# B&R Automation Studio project LABA4FINAL
Automation Studio 

## Configuration Real

### Task classes (Cpu.sw)
```
Cyclic#1:
  ncsdcctrl <- ncsdcctrl.prg
  SDCAxisCtr <- SDCAxisCtr.prg
  SDCAxisCt1 <- SDCAxisCtr1.prg
  SDCAxisCt2 <- SDCAxisCtr2.prg
DataObjects: Arnc0sys
NcDataObjects: AxisInit <- AxisInit.dob, gAxis03a <- gAxis03obj.gAxis03a.dob, gAxis03i <- gAxis03obj.gAxis03i.dob, AxisApt <- AxisApt.dob, gmcipvar <- GmcIpUserConfig.gmcipvar.dob, gmcipfun <- GmcIpUserConfig.gmcipfun.dob, gmcipfub <- GmcIpUserConfig.gmcipfub.dob, gmcipubr <- GmcIpUserConfig.gmcipubr.dob, gmcipusm <- GmcIpUserConfig.gmcipusm.dob, gmcipui <- GmcIpUserConfig.gmcipui.dob, gmcipus <- GmcIpUserConfig.gmcipus.dob, gmcipuc <- GmcIpUserConfig.gmcipuc.dob, gmcipsys <- GmcIpConfig.gmcipsys.dob, gmciplbr <- GmcIpConfig.gmciplbr.dob, gmcipcbr <- GmcIpConfig.gmcipcbr.dob, gmciplsm <- GmcIpConfig.gmciplsm.dob, gmcipcsm <- GmcIpConfig.gmcipcsm.dob, gmcipcfg <- GmcIpConfig.gmcipcfg.dob, gmcipiec <- GmcIpConfig.gmcipiec.dob, gmciplog <- GmcIpConfig.gmciplog.dob, gmcipesm <- GmcIpConfig.gmcipesm.dob, gmcipmxd <- GmcIpConfig.gmcipmxd.dob, gmcipmx <- GmcIpConfig.gmcipmx.dob, CncInit <- CncInit.dob, CncProg <- CncProg.dob, CncProg1 <- CncProg1.dob
Binaries: TCData, Acp10map1, acp10cfg, Acp10map, arconfig, User, Role, sysconf, iomap, asfw, ashwd, arnc0cfg, Arnc0map
Libraries: Acp10sdc, Library, Acp10man, Acp10_MC, sys_lib, brsystem, asstring, powerlnk, asieccon, AsMath, Arnc0man, DataObj, AsArLog, FileIO, AsArProf, AsMem, Runtime, astime, Acp10par, NcGlobal, asiotime
```

### IoMap.iom - 4PP065_0571_P74/IoMap.iom
```iecst
VAR_CONFIG
	Cyclic#1.gAxis03_DrvIf.iLifeCnt AT %IB."8I64xxxxxxx.00x-1".SDC_LifeCnt;
	Cyclic#1.gAxis03_DrvIf.iDrvOK AT %IX."8I64xxxxxxx.00x-1".ETAD_Input_Bool_02;
	Cyclic#1.gAxis03_DrvIf.oSetTime AT %QW."8I64xxxxxxx.00x-1".SDC_SetTime;
	Cyclic#1.gAxis03_DrvIf.oSetPos AT %QW."8I64xxxxxxx.00x-1".LFRD_Output;
	Cyclic#1.gAxis03_DiDoIf.iLifeCntDriveReady AT %IB."8I64xxxxxxx.00x-1".SDC_LifeCnt;
	Cyclic#1.gAxis03_DiDoIf.iLifeCntDriveEnable AT %IB."8I64xxxxxxx.00x-1".SDC_LifeCnt;
	Cyclic#1.gAxis03_DiDoIf.oDriveEnable AT %QX."8I64xxxxxxx.00x-1".CMDD_Output_Bool_00;
	Cyclic#1.gAxis03_ModuleOk AT %QX."8I64xxxxxxx.00x-1".CMDD_Output_Bool_01;
	Cyclic#1.gAxis03_ModuleOk AT %QX."8I64xxxxxxx.00x-1".CMDD_Output_Bool_02;
	Cyclic#1.gAxis03_ModuleOk AT %IX."8I64xxxxxxx.00x-1".ModuleOk;
	Cyclic#1.gAxis03_DiDoIf.oDriveEnable AT %QX."8I64xxxxxxx.00x-1".CMDD_Output_Bool_03;
	Cyclic#1.gAxis03_DiDoIf.iDriveReady AT %IX."8I64xxxxxxx.00x-1".ETAD_Input_Bool_02;
	::SDCAxisCtr:pwm_period AT %QW."X20MM4456".PeriodDurationPWM;
	::SDCAxisCtr:coil_pwm_value AT %QW."X20MM4456".PulseWidthCurrentPWM04;
	::SDCAxisCtr:axis_X.pwm_value AT %QW."X20MM4456".PulseWidthCurrentPWM01;
	::SDCAxisCtr:axis_X.reset_error AT %QX."X20MM4456".ClearError01;
	::SDCAxisCtr:axis_X.reset_counter AT %QX."X20MM4456".ResetCounter01;
	::SDCAxisCtr:axis_X.counter AT %IW."X20MM4456".Counter01;
	::SDCAxisCtr:axis_X.endswitch_a_reached AT %IX."X20MM4456".StatusInput03; (*Logical condition input 01=Motor 01:A*)
	::SDCAxisCtr:axis_X.endswitch_b_reached AT %IX."X20MM4456".StatusInput04; (*Logical condition input 02=Motor 01:B*)
	::SDCAxisCtr:coil_powered AT %IX."X20DI9371".DigitalInput01;
	::SDCAxisCt1:axis_Y.pwm_value AT %QW."X20MM4456".PulseWidthCurrentPWM02;
	::SDCAxisCt1:axis_Y.reset_error AT %QX."X20MM4456".ClearError02;
	::SDCAxisCt1:axis_Y.reset_counter AT %QX."X20MM4456".ResetCounter02;
	::SDCAxisCt1:axis_Y.counter AT %IW."X20MM4456".Counter02;
	::SDCAxisCt1:axis_Y.endswitch_a_reached AT %IX."X20MM4456".StatusInput07;
	::SDCAxisCt1:axis_Y.endswitch_b_reached AT %IX."X20MM4456".StatusInput08;
	::SDCAxisCt2:axis_Z.pwm_value AT %QW."X20MM4456".PulseWidthCurrentPWM03;
	::SDCAxisCt2:axis_Z.reset_error AT %QX."X20MM4456".ClearError03;
	::SDCAxisCt2:axis_Z.reset_counter AT %QX."X20MM4456".ResetCounter03;
	::SDCAxisCt2:axis_Z.counter AT %IW."X20MM4456".Counter03;
	::SDCAxisCt2:axis_Z.endswitch_a_reached AT %IX."X20MM4456".StatusInput11;
	::SDCAxisCt2:axis_Z.endswitch_b_reached AT %IX."X20MM4456".StatusInput12;
	::SDCAxisCt1:coil_powered AT %IX."X20DI9371".DigitalInput02;
	::SDCAxisCt2:coil_powered AT %IX."X20DI9371".DigitalInput03;
END_VAR
```

### Acp10map.ncm - 4PP065_0571_P74/Motion/Acp10map.ncm
```
NcMapping (NcSwId=Acp10, DisabledNodesAreHidden=False)
  NcObject gAxis03 (ModuleId=8I64xxxxxxx.00x-1, ModuleAddress=SDC_IF1.ST1, Type=ncAXIS, Channel=1, AcoposSimulation=Off, InitParameter=gAxis03i, AcoposParameter=gAxis03a, AdditionalData=CNC_Enabled="1" , Disabled=FALSE, ModuleDisabled=FALSE)
```

### Arnc0map.ncm - 4PP065_0571_P74/Motion/Arnc0map.ncm
```
NcMapping (NcSwId=Arnc0, DisabledNodesAreHidden=False)
  NcObject CNCsys (Type=ncCNCSYS, Channel=1, AcoposSimulation=Off, InitParameter=CncInit, Disabled=FALSE, ModuleDisabled=FALSE)
  NcObject CNC2 (Type=ncCNCSYS, Channel=2, AcoposSimulation=Off, Disabled=TRUE, ModuleDisabled=FALSE)
  NcObject CNC3 (Type=ncCNCSYS, Channel=3, AcoposSimulation=Off, Disabled=TRUE, ModuleDisabled=FALSE)
  NcObject CNC4 (Type=ncCNCSYS, Channel=4, AcoposSimulation=Off, Disabled=TRUE, ModuleDisabled=FALSE)
  NcObject CNC5 (Type=ncCNCSYS, Channel=5, AcoposSimulation=Off, Disabled=TRUE, ModuleDisabled=FALSE)
  NcObject CNC6 (Type=ncCNCSYS, Channel=6, AcoposSimulation=Off, Disabled=TRUE, ModuleDisabled=FALSE)
  NcObject CNC7 (Type=ncCNCSYS, Channel=7, AcoposSimulation=Off, Disabled=TRUE, ModuleDisabled=FALSE)
  NcObject CNC8 (Type=ncCNCSYS, Channel=8, AcoposSimulation=Off, Disabled=TRUE, ModuleDisabled=FALSE)
  NcObject CNC9 (Type=ncCNCSYS, Channel=9, AcoposSimulation=Off, Disabled=TRUE, ModuleDisabled=FALSE)
  NcObject CNC10 (Type=ncCNCSYS, Channel=10, AcoposSimulation=Off, Disabled=TRUE, ModuleDisabled=FALSE)
  NcObject CNC11 (Type=ncCNCSYS, Channel=11, AcoposSimulation=Off, Disabled=TRUE, ModuleDisabled=FALSE)
  NcObject CNC12 (Type=ncCNCSYS, Channel=12, AcoposSimulation=Off, Disabled=TRUE, ModuleDisabled=FALSE)
  NcObject CNC13 (Type=ncCNCSYS, Channel=13, AcoposSimulation=Off, Disabled=TRUE, ModuleDisabled=FALSE)
  NcObject CNC14 (Type=ncCNCSYS, Channel=14, AcoposSimulation=Off, Disabled=TRUE, ModuleDisabled=FALSE)
  NcObject CNC15 (Type=ncCNCSYS, Channel=15, AcoposSimulation=Off, Disabled=TRUE, ModuleDisabled=FALSE)
  NcObject CNC16 (Type=ncCNCSYS, Channel=16, AcoposSimulation=Off, Disabled=TRUE, ModuleDisabled=FALSE)
  NcObject CNC17 (Type=ncCNCSYS, Channel=17, AcoposSimulation=Off, Disabled=TRUE, ModuleDisabled=FALSE)
  NcObject CNC18 (Type=ncCNCSYS, Channel=18, AcoposSimulation=Off, Disabled=TRUE, ModuleDisabled=FALSE)
  NcObject CNC19 (Type=ncCNCSYS, Channel=19, AcoposSimulation=Off, Disabled=TRUE, ModuleDisabled=FALSE)
  NcObject CNC20 (Type=ncCNCSYS, Channel=20, AcoposSimulation=Off, Disabled=TRUE, ModuleDisabled=FALSE)
  NcObject CNC21 (Type=ncCNCSYS, Channel=21, AcoposSimulation=Off, Disabled=TRUE, ModuleDisabled=FALSE)
  NcObject CNC22 (Type=ncCNCSYS, Channel=22, AcoposSimulation=Off, Disabled=TRUE, ModuleDisabled=FALSE)
  NcObject CNC23 (Type=ncCNCSYS, Channel=23, AcoposSimulation=Off, Disabled=TRUE, ModuleDisabled=FALSE)
  NcObject CNC24 (Type=ncCNCSYS, Channel=24, AcoposSimulation=Off, Disabled=TRUE, ModuleDisabled=FALSE)
```

## Configuration Simulation

CPU , AutomationRuntime J4.25

### Task classes (Cpu.sw)
```
Cyclic#1 (cycle 100000 us, tolerance 0 us):
  SDCAxisCtr <- SDCAxisCtr.prg
DataObjects: Acp10sys
NcDataObjects: AxisApt <- AxisApt.dob, AxisInit <- AxisInit.dob, acp10etxen <- acp10etxen.dob
Binaries: TCData, ashwd, sysconf, asfw, arconfig, iomap, Acp10map, Acp10map1, arnc0cfg, acp10cfg
Libraries: AsIecCon, astime, Acp10sdc, Acp10man, Acp10par, NcGlobal, asstring, AsIOTime, Acp10_MC, brsystem, sys_lib, Runtime, Acp10sim, fileio, powerlnk, Library
```

### Hardware
```
PC_any : PC_any v1.1.0.0 (OrderNumber=PC)
  ConfigurationID = SDCAxis_Simulation
  Cyclic1Duration = 100000
  Cyclic1Tolerance = 0
  Cyclic2Duration = 200000
  Cyclic2Tolerance = 10000000
  Cyclic3Duration = 500000
  Cyclic3Tolerance = 10000000
  Cyclic4Duration = 1000000
  Cyclic4Tolerance = 10000000
  Cyclic5Duration = 2000000
  Cyclic5Tolerance = 10000000
  Cyclic6Duration = 3000000
  Cyclic6Tolerance = 12000000
  Cyclic7Duration = 4000000
  Cyclic7Tolerance = 12000000
  Cyclic8Duration = 5000000
  Cyclic8Tolerance = 30000000
```

## Logical view

### Global.var - Global variables
```iecst
VAR
	AxisX : ACP10AXIS_typ := (0);
	AxisX_EncIf : SdcEncIf16_typ := (0);
	AxisX_DrvIf : SdcDrvIf16_typ := (0);
	AxisX_DiDoIf : SdcDiDoIf_typ := (0);
	AxisX_HW : SdcHwCfg_typ := (0);
	AxisY : ACP10AXIS_typ := (0);
	AxisY_EncIf : SdcEncIf16_typ := (0);
	AxisY_DrvIf : SdcDrvIf16_typ := (0);
	AxisY_DiDoIf : SdcDiDoIf_typ := (0);
	AxisY_HW : SdcHwCfg_typ := (0);
	AxisZ : ACP10AXIS_typ := (0);
	AxisZ_EncIf : SdcEncIf16_typ := (0);
	AxisZ_DrvIf : SdcDrvIf16_typ := (0);
	AxisZ_DiDoIf : SdcDiDoIf_typ := (0);
	AxisZ_HW : SdcHwCfg_typ := (0);
	gAxis01 : ACP10AXIS_typ := (0);
	gAxis02 : ACP10AXIS_typ := (0);
	gAxisTest : ACP10AXIS_typ := (0);
	gAxisTest_HW : SdcHwCfg_typ := (0);
	gAxisTest_DrvIf : SdcDrvIf16_typ := (0);
	gAxisTest_DiDoIf : SdcDiDoIf_typ := (0);
	gAxisTest_ModuleOk : BOOL := 0;
	gAxis03 : ACP10AXIS_typ := (0);
	gAxis03_HW : SdcHwCfg_typ := (0);
	gAxis03_DrvIf : SdcDrvIf16_typ := (0);
	gAxis03_DiDoIf : SdcDiDoIf_typ := (0);
	gAxis03_ModuleOk : BOOL := 0;
	CNCsys : ARNC0CNC_typ;
END_VAR
```

### Package Logical/Libraries - Global libraries

### Library Logical/Libraries/Library (ANSIC)

#### Library.fun
```iecst
FUNCTION_BLOCK FB_Motor (*TODO: Add your comment here*) (*$GROUP=User,$CAT=User,$GROUPICON=User.png,$CATICON=User.png*)
	VAR_INPUT
		in : REAL;
	END_VAR
	VAR_OUTPUT
		out_w : REAL;
		out_phi : REAL;
	END_VAR
	VAR
		k_e : REAL;
		T_m : REAL;
		dt : REAL;
		integrator : FB_Integrator;
		integrator_phi : FB_Integrator;
	END_VAR
END_FUNCTION_BLOCK

FUNCTION_BLOCK FB_Integrator (*TODO: Add your comment here*) (*$GROUP=User,$CAT=User,$GROUPICON=User.png,$CATICON=User.png*)
	VAR_INPUT
		in : REAL;
		dt : REAL;
	END_VAR
	VAR_OUTPUT
		out : REAL;
	END_VAR
	VAR
		state : REAL := 0.0;
	END_VAR
END_FUNCTION_BLOCK

FUNCTION_BLOCK FB_Controller (* *) (*$GROUP=User,$CAT=User,$GROUPICON=User.png,$CATICON=User.png*)
	VAR_INPUT
		in : REAL;
	END_VAR
	VAR_OUTPUT
		out : REAL;
	END_VAR
	VAR
		k_i : REAL;
		sum : REAL;
		k_p : REAL;
		dt : REAL;
		max_abs_value : REAL;
		integrator : FB_Integrator;
		last_sum : REAL;
	END_VAR
END_FUNCTION_BLOCK

FUNCTION_BLOCK FB_Endswitch (*TODO: Add your comment here*) (*$GROUP=User,$CAT=User,$GROUPICON=User.png,$CATICON=User.png*)
	VAR_INPUT
		in : REAL;
		neg_value : REAL;
		pos_value : REAL;
	END_VAR
	VAR_OUTPUT
		neg_reached : BOOL;
		pos_reached : BOOL;
	END_VAR
END_FUNCTION_BLOCK

FUNCTION_BLOCK FB_Axis (*TODO: Add your comment here*) (*$GROUP=User,$CAT=User,$GROUPICON=User.png,$CATICON=User.png*)
	VAR_INPUT
		reset_error : BOOL;
		endswitch_a_reached : BOOL;
		endswitch_b_reached : BOOL;
		pwm_percentage : SINT;
	END_VAR
	VAR_OUTPUT
		reset_counter : BOOL;
		pwm_value : INT;
	END_VAR
	VAR_OUTPUT RETAIN
		counter : INT;
	END_VAR
	VAR_OUTPUT
		speed : REAL;
	END_VAR
	VAR
		last_counter : INT;
	END_VAR
END_FUNCTION_BLOCK
```

#### FB_Controller.c
```c
#include <bur/plctypes.h>
#ifdef __cplusplus
	extern "C"
	{
#endif
	#include "Library.h"
#ifdef __cplusplus
	};
#endif

void FB_Controller(struct FB_Controller* inst)
{
	REAL a = inst->in * inst->k_p;
	REAL b = inst->in * inst->k_i;
	inst->integrator.dt = inst->dt;
	inst->integrator.in = b;
	FB_Integrator(&inst->integrator);
	a = a > inst->max_abs_value ? inst->max_abs_value : a;
	a = a < -inst->max_abs_value ? -inst->max_abs_value : a;
	inst->sum = a + inst->integrator.out;
	inst->out = inst->sum;
	inst->out = inst->out > inst->max_abs_value ? inst->max_abs_value : inst->out;
	inst->out = inst->out < -inst->max_abs_value ? -inst->max_abs_value : inst->out;
	inst->last_sum = (inst->out - inst->sum);
	inst->integrator.state = inst->integrator.state + inst->last_sum;
}
```

#### FB_Endswitch.c
```c
#include <bur/plctypes.h>
#ifdef __cplusplus
	extern "C"
	{
#endif
	#include "Library.h"
#ifdef __cplusplus
	};
#endif
/* TODO: Add your comment here */
void FB_Endswitch(struct FB_Endswitch* inst)
{
	inst->pos_reached = inst->in >= inst->pos_value ? 1 : 0;
	inst->neg_reached = inst->in <= inst->neg_value ? 1 : 0;
}
```

### Data object Logical/AxisInit (Ax)

#### AxInitAcp10.ax
```
InitParameter (Version=3.13.1, NcSwId=ACP10)
  ACP10AXIS_typ:
    dig_in:
      level:
        reference = ncACTIV_HI
        pos_hw_end = ncACTIV_HI
        neg_hw_end = ncACTIV_HI
        trigger1 = ncACTIV_HI
        trigger2 = ncACTIV_HI
    encoder_if:
      parameter:
        count_dir = ncSTANDARD
        scaling:
          load:
            units = 3000
            rev_motor = 1
    limit:
      parameter:
        v_pos = 7500.0
        v_neg = 7500.0
        a1_pos = 10000.0
        a2_pos = 10000.0
        a1_neg = 10000.0
        a2_neg = 10000.0
        t_jolt = 0.0
        t_in_pos = 0.0
        pos_sw_end = 8388607
        neg_sw_end = -8388608
        ds_warning = 500.0
        ds_stop = 1000.0
        a_stop = 1.0E+30
        dv_stop = 0.0
        dv_stop_mode = ncOFF
    controller:
      mode = ncPOSITION
      position:
        kv = 10.0
        tn = 0.0
        t_predict = 0.04
        t_total = 0.04
        p_max = 10000.0
        i_max = 0.0
      speed:
        kv = 2.0
        tn = 0.0
        t_filter = 0.0
        isq_filter1:
          type = ncOFF
          a0 = 0.0
          a1 = 0.0
          b0 = 0.0
          b1 = 0.0
          b2 = 0.0
          c0_par_id = 0
          c1_par_id = 0
        isq_filter2:
          type = ncOFF
          a0 = 0.0
          a1 = 0.0
          b0 = 0.0
          b1 = 0.0
          b2 = 0.0
          c0_par_id = 0
          c1_par_id = 0
        isq_filter3:
          type = ncOFF
          a0 = 0.0
          a1 = 0.0
          b0 = 0.0
          b1 = 0.0
          b2 = 0.0
          c0_par_id = 0
          c1_par_id = 0
      uf:
        type = ncLINEAR
        auto_config = ncMOTOR_PAR
        u0 = 0.0
        un = 0.0
        fn = 50.0
        k_f_slip = 0.0
      ff:
        torque_load = 0.0
        torque_pos = 0.0
        torque_neg = 0.0
        kv_torque = 0.0
        inertia = 0.0
        t_filter_a = 0.0
    move:
      stop:
        parameter[0]:
          decel_ramp = ncA_LIMIT
          controller = ncON
        parameter[1]:
          decel_ramp = ncA_LIMIT
          controller = ncON
        parameter[2]:
          decel_ramp = ncA_LIMIT
          controller = ncON
        parameter[3]:
          decel_ramp = ncA_LIMIT
          controller = ncON
        quickstop:
          decel_ramp = ncA_LIMIT
        drive_error:
          decel_ramp = ncA_LIMIT
      homing:
        parameter:
          s = 0
          v_switch = 6000.0
          v_trigger = 2000.0
          a = 10000.0
          mode = ncDIRECT
          edge_sw = ncNEGATIVE
          start_dir = ncPOSITIVE
          trigg_dir = ncNEGATIVE
          ref_pulse = ncOFF
          fix_dir = ncOFF
          tr_s_block = 0.0
          torque_lim = 0.0
          ds_block = 0.0
          ds_stop = 0.0
      basis:
        parameter:
          v_pos = 4000.0
          v_neg = 4000.0
          a1_pos = 10000.0
          a2_pos = 10000.0
          a1_neg = 10000.0
          a2_neg = 10000.0
    message:
      text:
        parameter:
          format = ncBREAK
          columns = 80
          data_modul
```

### Program Logical/ncsdcctrl (IEC)

#### ncsdcctrlCyclic.st
```iecst
PROGRAM _CYCLIC

(* ### BEGIN gAxisTest ### *)

(* life counter emulation of digital inputs *)
 gAxisTest_DiDoIf.iLifeCntReference := gAxisTest_DiDoIf.iLifeCntReference + 1;
 gAxisTest_DiDoIf.iLifeCntNegHwEnd  := gAxisTest_DiDoIf.iLifeCntNegHwEnd  + 1;
 gAxisTest_DiDoIf.iLifeCntPosHwEnd  := gAxisTest_DiDoIf.iLifeCntPosHwEnd  + 1;

(* ### END gAxisTest ### *)

(* ### BEGIN gAxis03 ### *)

(* life counter emulation of digital inputs *)
 gAxis03_DiDoIf.iLifeCntReference := gAxis03_DiDoIf.iLifeCntReference + 1;
 gAxis03_DiDoIf.iLifeCntNegHwEnd  := gAxis03_DiDoIf.iLifeCntNegHwEnd  + 1;
 gAxis03_DiDoIf.iLifeCntPosHwEnd  := gAxis03_DiDoIf.iLifeCntPosHwEnd  + 1;

(* ### END gAxis03 ### *)

END_PROGRAM
```

#### ncsdcctrlInit.st
```iecst
PROGRAM _INIT

(* ### BEGIN gAxisTest ### *)

(* initialize variables *)
 gAxisTest_HW.DrvIf_Typ := ncSDC_DRVSERVO16;
 strcpy( ADR(gAxisTest_HW.DrvIf_Name[0]), ADR('gAxisTest_DrvIf') );
 gAxisTest_HW.DiDoIf_Typ := ncSDC_DIDO;
 strcpy( ADR(gAxisTest_HW.DiDoIf_Name[0]), ADR('gAxisTest_DiDoIf') );

(* force variable offset generation *)
 gAxisTest.size                      := gAxisTest.size;
 gAxisTest_DrvIf.iLifeCnt            := gAxisTest_DrvIf.iLifeCnt;
 gAxisTest_DiDoIf.iLifeCntDriveReady := gAxisTest_DiDoIf.iLifeCntDriveReady;
 gAxisTest_ModuleOk                  := gAxisTest_ModuleOk;

(* assign your hardware inputs here*)

(* gAxisTest_DiDoIf.iPosHwEnd  := gAxisTest_DiDoIf.iPosHwEnd;
 gAxisTest_DiDoIf.iNegHwEnd  := gAxisTest_DiDoIf.iNegHwEnd;
 gAxisTest_DiDoIf.iReference := gAxisTest_DiDoIf.iReference;
 *)

(* ### END gAxisTest ### *)

(* ### BEGIN gAxis03 ### *)

(* initialize variables *)
 gAxis03_HW.DrvIf_Typ := ncSDC_DRVSERVO16;
 strcpy( ADR(gAxis03_HW.DrvIf_Name[0]), ADR('gAxis03_DrvIf') );
 gAxis03_HW.DiDoIf_Typ := ncSDC_DIDO;
 strcpy( ADR(gAxis03_HW.DiDoIf_Name[0]), ADR('gAxis03_DiDoIf') );

(* force variable offset generation *)
 gAxis03.size                      := gAxis03.size;
 gAxis03_DrvIf.iLifeCnt            := gAxis03_DrvIf.iLifeCnt;
 gAxis03_DiDoIf.iLifeCntDriveReady := gAxis03_DiDoIf.iLifeCntDriveReady;
 gAxis03_ModuleOk                  := gAxis03_ModuleOk;

(* assign your hardware inputs here*)

(* gAxis03_DiDoIf.iPosHwEnd  := gAxis03_DiDoIf.iPosHwEnd;
 gAxis03_DiDoIf.iNegHwEnd  := gAxis03_DiDoIf.iNegHwEnd;
 gAxis03_DiDoIf.iReference := gAxis03_DiDoIf.iReference;
 *)

(* ### END gAxis03 ### *)

END_PROGRAM
```

- gmcipcbr.cnc (not shown)

### Data object Logical/GmcIpConfig/gmcipcfg (Cnc, version 3.13.0)

#### gmcipcfg.cnc
```
CONFIG:
  LANG_INCLUDE gmcipmxd (LangName=IEC-ST, DataObject=Yes, IfNotExist=Error, Scope=NC_GLOBAL, RequireFnIgnore=MXConvertOrient)
  XML_INCLUDE gmcipvar (IfNotExist=Warn)
  XML_INCLUDE gmcipfun (IfNotExist=Warn)
  XML_INCLUDE gmcipfub (IfNotExist=Warn)
  MPQUEUE (NumPackets=200, LookaheadMinBlocks=5, LookaheadMaxBlocks=20, LookaheadMode=any, MaxPathJobs=256)
  MONITOR (MaxPathStackEvents=1024)
  MPLOG (MaxBuffers=10, MinBuffers=4, EarlyCircleBufferLookahead=2, DefaultBufferSize=131072, TaskCycleDelay=1, FileDevice=mplog*, MaxLogFiles=20, MaxLogFileSize=1048576, CopyLineTextMaxChars=80)
  AXES (StandardCNCAxes=Yes)
  FUBOutputs:
    FUBOutput PLCOpen:
      ERROR (condition=$Error == 1)
      BUSY (condition=$Busy == 1)
    FUBOutput BuR:
      ERROR (condition=$status != 65535 && $status != 0)
      BUSY (condition=$status == 65535)
  FUNCTIONS:
    FUNC LEN (DeclareName=__LEN, AlwaysDeclare=Yes, RetType=INT)
      ARG IN (Type=STRING)
    FUNC LEFT (DeclareName=__LEFT, AlwaysDeclare=Yes, RetType=STRING, RetRef=Yes)
      ARG IN (Type=STRING)
      ARG L (Type=INT)
    FUNC RIGHT (DeclareName=__RIGHT, AlwaysDeclare=Yes, RetType=STRING, RetRef=Yes)
      ARG IN (Type=STRING)
      ARG L (Type=INT)
    FUNC MID (DeclareName=__MID, AlwaysDeclare=Yes, RetType=STRING, RetRef=Yes)
      ARG IN (Type=STRING)
      ARG L (Type=INT)
      ARG P (Type=INT)
    FUNC CONCAT (DeclareName=__CONCAT, AlwaysDeclare=Yes, RetType=STRING, RetRef=Yes)
      ARG IN1 (Type=STRING)
      ARG IN2 (Type=STRING)
    FUNC INSERT (DeclareName=__INSERT, AlwaysDeclare=Yes, RetType=STRING, RetRef=Yes)
      ARG IN1 (Type=STRING)
      ARG IN2 (Type=STRING)
      ARG P (Type=INT)
    FUNC DELETE (DeclareName=__DELETE, AlwaysDeclare=Yes, RetType=STRING, RetRef=Yes)
      ARG IN (Type=STRING)
      ARG L (Type=INT)
      ARG P (Type=INT)
    FUNC REPLACE (DeclareName=__REPLACE, AlwaysDeclare=Yes, RetType=STRING, RetRef=Yes)
      ARG IN1 (Type=STRING)
      ARG IN2 (Type=STRING)
      ARG L (Type=INT)
      ARG P (Type=INT)
    FUNC FIND (DeclareName=__FIND, AlwaysDeclare=Yes, RetType=INT)
      ARG IN1 (Type=STRING)
      ARG IN2 (Type=STRING)
  XML_INCLUDE gmcipuc (IfNotExist=Warn)
```

- Data object Logical/GmcIpConfig/gmcipcsm (Cnc, version 3.13.0) (no source held here)

### gmcipesm.cnc
```
Root (LangModule=ailgcode, Version=1.0)
  AILHeader = def ip_global BOOL  __CANCEL_RND 
    def ip_global BOOL  __C2_SPLINE_ACTIVE 
    def ip_global LREAL __RNDM_RADIUS 
    def ip_global LREAL __CSPLINE_CHORD_ERROR 
    def ip_global DINT __SET_GXX_ACTIVE 
    def ip_global DINT __SET_GXX_REACTIVATE 
    def ip_global DINT __SET_GXX_CALL_CNT 
    def ip_global REAL __VAR1 
    def ip_global DINT __ACTIVE_MIRROR 

    sub OnProgStart
      %__CANCEL_RND = 0;
      %__RNDM_RADIUS = 0.0;
      %__C2_SPLINE_ACTIVE = 0;
      %__CSPLINE_CHORD_ERROR = 0.001;
      %__SET_GXX_ACTIVE = 0;
      %__SET_GXX_REACTIVATE = 0;
      %__SET_GXX_CALL_CNT = 0;
      %__ACTIVE_MIRROR = 20;
    endsub

    sub EndSplineSection
      
      if (%__C2_SPLINE_ACTIVE)
        `T:GCodes,G802`(:"bc_par":1 :);
        %__C2_SPLINE_ACTIVE = 0;
        
        DispatchMPList(::);
      endif
    endsub
    sub WriteZpTable
      
      #next_motion.Command = MPCMD_SET_ZP_TABLE;
      #next_motion.Data.SetZeroPtTable.ZpRecIdx = $[1];
      #next_motion.Data.SetZeroPtTable.ZpOffset[0] = $[2];
      #next_motion.Data.SetZeroPtTable.ZpOffset[1] = $[3];
      #next_motion.Data.SetZeroPtTable.ZpOffset[2] = $[4];
      PushPacket(::);
      DispatchMPList(::);
    endsub

    sub ReactivateGxx
      
      
      if (%__SET_GXX_CALL_CNT != 0)
          if (%__SET_GXX_REACTIVATE == 1)
            `T:GCodes,G54`(::);
             DispatchMPList(::);
             #sys_vars.ZP = %__SET_GXX_REACTIVATE;
          elif (%__SET_GXX_REACTIVATE == 2)
            `T:GCodes,G55`(::);
             DispatchMPList(::);
             #sys_vars.ZP = %__SET_GXX_REACTIVATE;
          elif (%__SET_GXX_REACTIVATE == 3)
            `T:GCodes,G56`(::);
             DispatchMPList(::);
             #sys_vars.ZP = %__SET_GXX_REACTIVATE;
          elif (%__SET_GXX_REACTIVATE == 4)
            `T:GCodes,G57`(::);
             DispatchMPList(::);
             #sys_vars.ZP = %__SET_GXX_REACTIVATE;
          elif (%__SET_GXX_REACTIVATE == 5)
            `T:GCodes,G58`(::);
             DispatchMPList(::);
             #sys_vars.ZP = %__SET_GXX_REACTIVATE;
          elif (%__SET_GXX_REACTIVATE == 6)
            `T:GCodes,G59`(::);
             DispatchMPList(::);
             #sys_vars.ZP = %__SET_GXX_REACTIVATE;
          endif
          %__SET_GXX_REACTIVATE = 0;
          %__SET_GXX_CALL_CNT = 0;
      endif
    endsub (Append=Yes)
  BuiltInProcs:
    RESET_G54 = WriteZpTable(:1, 0.0, 0.0, 0.0:); (MinArgs=0, MaxArgs=0)
    RESET_G55 = WriteZpTable(:2, 0.0, 0.0, 0.0:); (MinArgs=0, MaxArgs=0)
    RESET_G56 = WriteZpTable(:3, 0.0, 0.0, 0.0:); (MinArgs=0, MaxArgs=0)
    RESET_G57 = WriteZpTable(:4, 0.0, 0.0, 0.0:); (MinArgs=0, MaxArgs=0)
    RESET_G58 = WriteZpTable(:5, 0.0, 0.0, 0.0:); (MinArgs=0, MaxArgs=0)
    RESET_G59 = WriteZpTable(:6, 0.0, 0.0, 0.0:); (MinArgs=0, MaxArgs=0)
    SET_G54 = WriteZpTable(:1, $[1], $[2], $[3]:);
      %_CNC.move_cmd_mode = MPCMD_LIN_INTPOL;
      %__SET_GXX_ACTIVE = 1;
      %__SET_GXX_REACTIVATE = 0;
      %__SET_GXX_CALL_CNT = 0;		
      
      `T:GCodes,G54`(::);
      #sys_vars.ZP = 1; (MinArgs=3, MaxArgs=3)
    SET_G55 = WriteZpTable(:2, $[1], $[2], $[3]:);
      %_CNC.move_cmd_mode = MPCMD_LIN_INTPOL;
      %__SET_GXX_ACTIVE = 2;
      %__SET_GXX_REACTIVATE = 0;
      %__SET_GXX_CALL_CNT = 0;		
      `T:GCodes,G55`(::);
      #sys_vars.ZP = 2; (MinArgs=3, MaxArgs=3)
    SET_G56 = WriteZpTable(:3, $[1], $[2], $[3]:);
      %_CNC.move_cmd_mode = MPCMD_LIN_INTPOL;
      %__SET_GXX_ACTIVE = 3;
      %__SET_GXX_REACTIVATE = 0;
      %__SET_GXX_CALL_CNT = 0;		
      `T:GCodes,G56`(::);
      #sys_vars.ZP = 3; (MinArgs=3, MaxArgs=3)
    SET_G57 = WriteZpTable(:4, $[1], $[2], $[3]:);
      %_CNC.move_cmd_mode = MPCMD_LIN_INTPOL;
      %__SET_GXX_ACTIVE = 4;
      %__SET_GXX_REACTIVATE = 0;
      %__SET_GXX_CALL_CNT = 0;		
      `T:GCodes,G57`(::);
      #sys_vars.ZP = 4; (MinArgs=3, MaxArgs=3)
    SET_G58 = WriteZpTable(:5, $[1], $[2], $[3]:);
      %_CNC.move_cmd_mode = MPCMD_LIN_INTPOL;
      %__SET_GXX_ACTIVE = 5;
      %__SET_GXX_REACTIVATE = 0;
      %__SET_GXX_CALL_CNT = 0;		
      `T:GCodes,G58`(::);
      #sys_vars.ZP = 5; (MinArgs=3, MaxArgs=3)
    SET_G59 = WriteZpTable(:6, $[1], $[2], $[3]:);
      %_CNC.move_cmd_mode = MPCMD_LIN_INTPOL;
      %__SET_GXX_ACTIVE = 6;
      %__SET_GXX_REACTIVATE = 0;
      %__SET_GXX_CALL_CNT = 0;		
      `T:GCodes,G59`(::);
      #sys_vars.ZP = 6; (MinArgs=3, MaxArgs=3)
    RESET_MIRROR = `T:GCodes,G20`(::); (MinArgs=0, MaxArgs=0)
  PVMacros:
    WORKFRAME $WFRAME (ArrayDims=0)
      SET = `T:BuiltInProcs,RESET_SCALING`(::);
        #next_motion.Data.Frame.Data = ${EXPR};
        #next_motion.Command = MPCMD_W_FRAME;
        PushPacket(::); (Inline=Yes)
    WORKFRAME_ADD $WFRAME_ADD (ArrayDims=0)
      SET = `T:BuiltInProcs,RESET_SCALING`(::);
        #next_motion.Data.Frame.Data = ${EXPR};
        #next_motion.Command = MPCMD_W_FRAME_ADD;
        PushPacket(::); (Inline=Yes)
  GCodes:
    G_INIT_ESM = ReactivateGxx(::); (GNum=-5, AutoPush=Yes, Eval=First, Inline=No, GenerateIfGroups=1,1000)
    G_MODAL (GNum=-1, AutoPush=Yes, Group=1000, Eval=Normal, IgnoreIfNoArgs=Yes)
      Arg (ref=dest, MinCount=0, MaxCount=NumAxes, NameType=AXISREF, DataType=PositionValue, WriteOpts=#:u?)
      Arg (ref=center, MinCount=0, MaxCount=3, NameType=InterpolParam, DataType=PositionValue, WriteOpts=#:u?)
      Arg (ref=circlept, MinCount=0, MaxCount=3, NameType=CirclePointParam, DataType=PositionValue, WriteOpts=#:u?)
      Arg (ref=angle, MinCount=0, MaxCount=1, NameType=RotationAngleSpecifier, DataType=RotationAngle, WriteOpts=#:u?)
      Arg (ref=radius, MinCount=0, MaxCount=1, NameType=RadiusSpecifier, DataType=RadiusValue, WriteOpts=#:u?)
    G00 = %_CNC.move_cmd_mode = MPCMD_RAPID_MOVE_INTPOL;
      #sys_vars.modal_grp1_set = 1;
      EndSplineSection(::); (GNum=0, Group=1,50, Inline=Yes, Eval=Early)
    G01 = %_CNC.move_cmd_mode = MPCMD_LIN_INTPOL;
      #sys_vars.modal_grp1_set = 1;
      EndSplineSection(::); (GNum=1, Group=1,50, Inline=Yes, Eval=Early)
    G02 = %_CNC.move_cmd_mode = MPCMD_CIRC_INTPOL_CW;
      #sys_vars.modal_grp1_set = 1;
      EndSplineSection(::); (GNum=2, Group=1,51, Inline=Yes, Eval=Early)
    G03 = %_CNC.move_cmd_mode = MPCMD_CIRC_INTPOL_CCW;
      #sys_vars.modal_grp1_set = 1;
      EndSplineSection(::); (GNum=3, Group=1,51, Inline=Yes, Eval=Early)
    G20 = #next_motion.Command = MPCMD_MIRRORING;
      #next_motion.Data.I4_value = 20;
      %__ACTIVE_MIRROR = #next_motion.Data.I4_value;
      PushPacket(::); (GNum=20, Group=3)
    G20.1 (GNum=20.1, Alias=MIRROR, Group=3)
      Arg (DataType=AXISREF, ref=axis1, MinCount=0, MaxCount=1)
      Arg (DataType=EqString, ref=eq, MinCount=0, MaxCount=1)
      Arg (DataType=FLOAT, ref=dummy_pos1, MinCount=0, MaxCount=1)
      Arg (DataType=AXISREF, ref=axis2, MinCount=0, MaxCount=1)
      Arg (DataType=EqString, ref=eq, MinCount=0, MaxCount=1)
      Arg (DataType=FLOAT, ref=dummy_pos2, MinCount=0, MaxCount=1)
    G20.2 (GNum=20.2, Alias=AMIRROR, Group=3)
      Arg (DataType=AXISREF, ref=axis1, MinCount=1, MaxCount=1)
      Arg (DataType=EqString, ref=eq, MinCount=0, MaxCount=1)
      Arg (DataType=FLOAT, ref=dummy_pos1, MinCount=0, MaxCount=1)
      Arg (DataType=AXISREF, ref=axis2, MinCount=0, MaxCount=1)
      Arg (DataType=EqString, ref=eq, MinCount=0, MaxCount=1)
      Arg (DataType=FLOAT, ref=dummy_pos2, MinCount=0, MaxCount=1)
    G21 = #next_motion.Command = MPCMD_MIRRORING;
      #next_motion.Data.I4_value = 21;
      %__ACTIVE_MIRROR = #next_motion.Data.I4_value;
      PushPacket(::); (GNum=21, Group=3)
    G22 = #next_motion.Command = MPCMD_MIRRORING;
      #next_motion.Data.I4_value = 22;
      %__ACTIVE_MIRROR = #next_motion.Data.I4_value;
      PushPacket(::); (GNum=22, Group=3)
    G23 = #next_motion.Command = MPCMD_MIRRORING;
      #next_motion.Data.I4_value = 23;
      %__ACTIVE_MIRROR = #next_motion.Data.I4_value;
      PushPacket(::); (GNum=23, Group=3)
    G25.1 (GNum=25.1, Group=11, Alias=RNDM)
      Arg (NameType=EqString, DataType=TangArcRadius, ref=radius)
    G25.2 (GNum=25.2, Group=11, Alias=RND)
      Arg (NameType=EqString, DataType=TangArcRadius, ref=radius)
    G53 = #next_motion.Command = MPCMD_ABS_ZP_SHIFT;
      #next_motion.Data.AbsZeroPtShift.ZpRecIdx = 0;
      PushPacket(::);
      #sys_vars.ZP = 0;
      
      %__SET_GXX_REACTIVATE = %__SET_GXX_ACTIVE;
      %__SET_GXX_CALL_CNT = 0; (GNum=53, Group=6, AllowGroups=8,19,21,100,101,102,103)
    G92 (GNum=92, Group=21, ResetArgs=Yes, AllowGroups=6,8,19,32,100,101,102,103)
      Arg (NameType=AXISREF, DataType=PositionValue, ref=offset, MinCount=0, MaxCount=NumAxes, WriteOpts=#:u?)
      Arg (NameType=RotationAngleSpecifier, DataType=RotationAngle, ref=h_rot, MinCount=0, MaxCount=1, WriteOpts=#:u?, DenyArgs=3,4,5)
      Arg (NameType=EulerAngleName, DataType=RotationAngle, ref=e_rot, MinCount=0, MaxCount=3, WriteOpts=#:u?, DenyArgs=2,4,5)
      Arg (NameType=RPYAngleName, DataType=RotationAngle, ref=rpy_rot, MinCount=0, MaxCount=3, WriteOpts=#:u?, DenyArgs=2,3,5)
      Arg (NameType=RotaryVectorName, DataType=RotaryVector, ref=matrix, MinCount=0, MaxCount=3, WriteOpts=#:u?, DenyArgs=2,3,4)
    G92.1 (GNum=92.1, Group=21, ALIAS=SCALE, AliasIsPattern=Yes)
      Arg (DataType=FLOAT, ref=factor, MinCount=0, MaxCount=1)
    G92.2 (GNum=92.2, Group=21, ALIAS=ASCALE, AliasIsPattern=Yes)
      Arg (DataType=FLOAT, ref=factor, MinCount=1, MaxCount=1)
    G492 (GNum=492, Group=490, Alias=TRANS, AllowGroups=9999)
      Arg (NameType=AXISREF, DataType=PositionValue, ref=offsets, MinCount=0, MaxCount=NumAxes, WriteOpts=#:)
    G494 (GNum=494, Group=490, Alias=ROT, AllowGroups=9999, MinArgs=0, MaxArgs=1)
      Arg RPLArgPrefix (DataType=FLOAT, ref=rpl_value, MinCount=0, MaxCount=1, DenyArgs=offsets)
      Arg (NameType=AXISREF, DataType=PositionValue, ref=offsets, MinCount=0, MaxCount=NumAxes, DenyArgs=rpl_value, WriteOpts=#:)
    G500 = %__SET_GXX_REACTIVATE = 0;
       %__SET_GXX_ACTIVE = 0;
       %__SET_GXX_CALL_CNT = 0;
      `T:GCodes,G53`(::); (GNum=500, Group=6, AllowGroups=8,19,21,100,101,102,103)
    G804 = if (!%__C2_SPLINE_ACTIVE)
         
        `T:GCodes,G801`(:"seg_type":"CE", "seg_par":%__CSPLINE_CHORD_ERROR, "bc_par":1 :);
        %__C2_SPLINE_ACTIVE = 1;
        
        DispatchMPList(::);
        
        %_CNC.move_cmd_mode = MPCMD_LIN_INTPOL;
      endif (GNum=804, Alias=CSPLINE)
```

### Data object Logical/GmcIpConfig/gmcipiec (Cnc, version 3.13.0)

#### gmcipiec.cnc
```
Root (LangModule=ailgcode, Version=1.0)
  AxesSpec
  PrimTypes (PatternSuffix=:[^\d\w$#])
    BOOL (BRType=BOOL)
    STRING (BRType=STRING)
    WSTRING (BRType=WSTRING)
    TIME (BRType=TIME)
    SINT (BRType=SINT)
    INT (BRType=INT)
    DINT (BRType=DINT)
    USINT (BRType=USINT)
    UINT (BRType=UINT)
    UDINT (BRType=UDINT)
    REAL (BRType=REAL)
    LREAL (BRType=LREAL)
    DATE (BRType=DATE)
    DATE_AND_TIME (BRType=DATE_AND_TIME)
    DT (BRType=DT)
    TIME_OF_DAY (BRType=TIME_OF_DAY)
    TOD (BRType=TIME_OF_DAY)
    BYTE (BRType=BYTE)
    WORD (BRType=WORD)
    DWORD (BRType=DWORD)
  BuiltInProcs:
    SetCyclicId = #job->group_id = $[1]; (MinArgs=1, MaxArgs=1, Eval=Early)
    WaitForCyclic = if ( Defined(:$[1]:) ) 
        WaitForCyclicGroups(:${*}:);  
      else
        WaitForCyclicJob(:#last_job_id:);
      endif (MinArgs=0, MaxArgs=*)
    REPORT (MinArgs=2, MaxArgs=2)
      Arg (ref=id, DataType=INT)
      Arg (ref=msg, DataType=STRING)
    WARN (MinArgs=2, MaxArgs=2)
      Arg (ref=id, DataType=INT)
      Arg (ref=msg, DataType=STRING)
    HALT (MinArgs=2, MaxArgs=2)
      Arg (ref=id, DataType=INT)
      Arg (ref=msg, DataType=STRING)
    ERROR (MinArgs=2, MaxArgs=2)
      Arg (ref=id, DataType=INT)
      Arg (ref=msg, DataType=STRING)
    LOADBG (MinArgs=1, MaxArgs=1)
      Arg (ref=filename, DataType=STRING)
    LOAD (MinArgs=1, MaxArgs=1)
      Arg (ref=filename, DataType=STRING)
    UNLOAD (MinArgs=1, MaxArgs=1)
      Arg (ref=filename, DataType=STRING)
    EXEC (MinArgs=1, MaxArgs=5)
      Arg (ref=filename, DataType=STRING)
      Arg (ref=arguments, DataType=ANY_DATA)
      Arg (ref=langId, DataType=INT)
      Arg (ref=block, DataType=INT, MinCount=0, MaxCount=1, DenyArgs=5, WriteOpts=:)
      Arg (ref=line, DataType=INT, MinCount=0, MaxCount=1, DenyArgs=4, WriteOpts=:)
    EXEC_RPC (MinArgs=2, MaxArgs=4)
      Arg (ref=filename, DataType=STRING)
      Arg (ref=arguments, DataType=ANY_DATA)
      Arg (ref=langId, DataType=INT)
      Arg (ref=rpc, DataType=ANY_DATA, MinCount=1, MaxCount=1)
    EVAL (MinArgs=1, MaxArgs=2)
      Arg (ref=expression, DataType=STRING)
      Arg (ref=langId, DataType=INT)
    PUSH_PACKET = PushPacket(::);
    PUSH_PACKET_CMD (MinArgs=1, MaxArgs=2)
      Arg (ref=cmd, DataType=INT)
      Arg (ref=data, DataType=ANY_DATA)
    DISPATCH_AND_WAIT (MinArgs=1, MaxArgs=1)
      Arg (ref=cmd, DataType=INT)
    START_PACKET_LIST = #inhibit_mp_list_dispatch = 1;
    END_PACKET_LIST = #inhibit_mp_list_dispatch = 0;
    LOG_INFO (MinArgs=1, MaxArgs=1)
      Arg (ref=msg, DataType=STRING)
    SET_BLOCK_NUMBER = SetCurBlockNr(:$[1]:); (MinArgs=1, MaxArgs=1)
    SBLOF_PATH = #next_motion.Command = MPCMD_SBL_PATH_INHIBIT;
      PushPacket(::);
    SBLON_PATH = #next_motion.Command = MPCMD_SBL_PATH_RELEASE;
      PushPacket(::);
  BuiltInFns:
    ABS = Abs(:$[1]:) (ReturnType=ANY_NUM, ArgType1=ANY_NUM, Inline=Yes)
    SIN = RSin(:$[1]:) (ReturnType=ANY_REAL, ArgType1=ANY_REAL, Inline=Yes)
    COS = RCos(:$[1]:) (ReturnType=ANY_REAL, ArgType1=ANY_REAL, Inline=Yes)
    TAN = RTan(:$[1]:) (ReturnType=ANY_REAL, ArgType1=ANY_REAL, Inline=Yes)
    ASIN = RASin(:$[1]:) (ReturnType=ANY_REAL, ArgType1=ANY_REAL, Inline=Yes)
    ACOS = RACos(:$[1]:) (ReturnType=ANY_REAL, ArgType1=ANY_REAL, Inline=Yes)
    ATAN = RATan(:$[1]:) (ReturnType=ANY_REAL, ArgType1=ANY_REAL, Inline=Yes)
    SQRT = Sqrt(:$[1]:) (ReturnType=ANY_REAL, ArgType1=ANY_REAL, Inline=Yes)
    LN = Ln(:$[1]:) (ReturnType=ANY_REAL, ArgType1=ANY_REAL, Inline=Yes)
    EXP = Exp(:$[1]:) (ReturnType=ANY_REAL, ArgType1=ANY_REAL, Inline=Yes)
    LOG = Log(:$[1]:) (ReturnType=ANY_REAL, ArgType1=ANY_REAL, Inline=Yes)
    EXPT = Pow(:$[1],$[2]:) (ReturnType=ANY_REAL, ArgType1=ANY_REAL, ArgType2=ANY_NUM, Inline=Yes)
    TRUNC = ToInt(:Fix(:$[1]:):) (ReturnType=IEC_INT, ArgType1=FLOAT, Inline=Yes)
    ADR = Adr(:\$[1]:) (ReturnType=IEC_UDINT, ArgType1=ANY_DATA, Inline=Yes)
    REF = \$[1] (ReturnType=ANY_DATA, ArgType1=ANY_DATA, Inline=Yes)
    SIZEOF = Sizeof(:\$[1]:) (ReturnType=IEC_UINT, NumArgs=1, Inline=Yes)
    LIMIT (ReturnType=ANY_NUM, Inline=No)
      Arg (ref=MIN, DataType=ANY_NUM)
      Arg (ref=IN, DataType=ANY_NUM)
      Arg (ref=MAX, DataType=ANY_NUM)
    MIN (ReturnType=ANY_NUM, Inline=No)
      Arg (ref=IN1, DataType=ANY_NUM)
      Arg (ref=IN2, DataType=ANY_NUM)
    MAX (ReturnType=ANY_NUM, Inline=No)
      Arg (ref=IN1, DataType=ANY_NUM)
      Arg (ref=IN2, DataType=ANY_NUM)
    ROL = BitRotL(:$[1],$[2]:) (ReturnType=ANY_NUM, ArgType1=ANY_NUM, ArgType2=IEC_SINT)
    ROR = BitRotR(:$[1],$[2]:) (ReturnType=ANY_NUM, ArgType1=ANY_NUM, ArgType2=IEC_SINT)
    SHR = BitShR(:$[1],$[2]:) (ReturnType=ANY_NUM, ArgType1=ANY_NUM, ArgType2=IEC_SINT)
    SHL = BitShL(:$[1],$[2]:) (ReturnType=ANY_NUM, ArgType1=ANY_NUM, ArgType2=IEC_SINT)
    BIT_TST = AsBitTst(:$[1],$[2]:) (ReturnType=ANY_NUM, ArgType1=ANY_NUM, ArgType2=IEC_SINT)
    BIT_SET = AsBitSet(:$[1],$[2]:) (ReturnType=ANY_NUM, ArgType1=ANY_NUM, ArgType2=IEC_SINT)
    BIT_CLR = AsBitClr(:$[1],$[2]:) (ReturnType=ANY_NUM, ArgType1=ANY_NUM, ArgType2=IEC_SINT)
    TO_BOOL = ToBool(:$[1]:) (ReturnType=IEC_BOOL, ArgType1=ANY_DATA, Inline=Yes)
    TO_USINT = ToUInt(:$[1],1:) (ReturnType=IEC_USINT, ArgType1=ANY_DATA, Inline=Yes)
    TO_BYTE = ToUInt(:$[1],1:) (ReturnType=IEC_BYTE, ArgType1=ANY_DATA, Inline=Yes)
    TO_SINT = ToInt(:$[1],1:) (ReturnType=IEC_SINT, ArgType1=ANY_DATA, Inline=Yes)
    TO_UINT = ToUInt(:$[1],2:) (ReturnType=IEC_UINT, ArgType1=ANY_DATA, Inline=Yes)
    TO_WORD = ToUInt(:$[1],2:) (ReturnType=IEC_WORD, ArgType1=ANY_DATA, Inline=Yes)
    TO_INT = ToInt(:$[1],2:) (ReturnType=IEC_INT, ArgType1=ANY_DATA, Inline=Yes)
    TO_UDINT = ToUInt(:$[1]:) (ReturnType=IEC_UDINT, ArgType1=ANY_DATA, Inline=Yes)
    TO_DWORD = ToUInt(:$[1]:) (ReturnType=IEC_DWORD, ArgType1=ANY_DATA, Inline=Yes)
    TO_DINT = ToInt(:$[1]:) (ReturnType=IEC_DINT, ArgType1=ANY_DATA, Inline=Yes)
    TO_TIME = ToTime(:$[1]:) (ReturnType=IEC_TIME, ArgType1=ANY_DATA, Inline=Yes)
    TO_DT = ToDT(:$[1]:) (ReturnType=IEC_DT, ArgType1=ANY_DATA, Inline=Yes)
    TO_DATE_AND_TIME = ToDT(:$[1]:) (ReturnType=IEC_DT, ArgType1=ANY_DATA, Inline=Yes)
    TO_TOD = ToTOD(:$[1]:) (ReturnType=IEC_TOD, ArgType1=ANY_DATA, Inline=Yes)
    TO_TIME_OF_DAY = ToTOD(:$[1]:) (ReturnType=IEC_TOD, ArgType1=ANY_DATA, Inline=Yes)
    TO_DATE = ToDate(:$[1]:) (ReturnType=IEC_DATE, ArgType1=ANY_DATA, Inline=Yes)
    TO_REAL = ToFloat(:$[1]:) (ReturnType=IEC_REAL, ArgType1=ANY_DATA, Inline=Yes)
    TO_LREAL = ToLReal(:$[1]:) (ReturnType=IEC_LREAL, ArgType1=ANY_DATA, Inline=Yes)
    TO_STRING = ToString(:$[1]:) (ReturnType=IEC_STRING, ArgType1=ANY_DATA, Inline=Yes)
    TO_WSTRING = ToWString(:$[1]:) (ReturnType=IEC_WSTRING, ArgType1=ANY_DATA, Inline=Yes)
    USINT_TO_BOOL = ToBool(:$[1]:) (ReturnType=IEC_BOOL, ArgType1=IEC_USINT, Inline=Yes)
    SINT_TO_BOOL = ToBool(:$[1]:) (ReturnType=IEC_BOOL, ArgType1=IEC_SINT, Inline=Yes)
    UINT_TO_BOOL = ToBool(:$[1]:) (ReturnType=IEC_BOOL, ArgType1=IEC_UINT, Inline=Yes)
    INT_TO_BOOL = ToBool(:$[1]:) (ReturnType=IEC_BOOL, ArgType1=IEC_INT, Inline=Yes)
    UDINT_TO_BOOL = ToBool(:$[1]:) (ReturnType=IEC_BOOL, ArgType1=IEC_UDINT, Inline=Yes)
    DINT_TO_BOOL = ToBool(:$[1]:) (ReturnType=IEC_BOOL, ArgType1=IEC_DINT, Inline=Yes)
    REAL_TO_BOOL = ToBool(:$[1]:) (ReturnType=IEC_BOOL, ArgType1=IEC_REAL, Inline=Yes)
    LREAL_TO_BOOL = ToBool(:$[1]:) (ReturnType=IEC_BOOL, ArgType1=IEC_LREAL, Inline=Yes)
    TIME_TO_BOOL = ToBool(:$[1]:) (ReturnType=IEC_BOOL, ArgType1=IEC_TIME, Inline=Yes)
    DT_TO_BOOL = ToBool(:$[1]:) (ReturnType=IEC_BOOL, ArgType1=IEC_DT, Inline=Yes)
    TOD_TO_BOOL = ToBool(:$[1]:) (ReturnType=IEC_BOOL, ArgType1=IEC_TOD, Inline=Yes)
    BYTE_TO_BOOL = ToBool(:$[1]:) (ReturnType=IEC_BOOL, ArgType1=IEC_BYTE, Inline=Yes)
    WORD_TO_BOOL = ToBool(:$[1]:) (ReturnType=IEC_BOOL, ArgType1=IEC_WORD, Inline=Yes)
    DWORD_TO_BOOL = ToBool(:$[1]:) (ReturnType=IEC_BOOL, ArgType1=IEC_DWORD, Inline=Yes)
    BOOL_TO_USINT = ToUInt(:$[1],1:) (ReturnType=IEC_USINT, ArgType1=IEC_BOOL, Inline=Yes)
    SINT_TO_USINT = ToUInt(:$[1],1:) (ReturnType=IEC_USINT, ArgType1=IEC_SINT, Inline=Yes)
    UINT_TO_USINT = ToUInt(:$[1],1:) (ReturnType=IEC_USINT, ArgType1=IEC_UINT, Inline=Yes)
    INT_TO_USINT = ToUInt(:$[1],1:) (ReturnType=IEC_USINT, ArgType1=IEC_INT, Inline=Yes)
    UDINT_TO_USINT = ToUInt(:$[1],1:) (ReturnType=IEC_USINT, ArgType1=IEC_UDINT, Inline=Yes)
    DINT_TO_USINT = ToUInt(:$[1],1:) (ReturnType=IEC_USINT, ArgType1=IEC_DINT, Inline=Yes)
    REAL_TO_USINT = ToUInt(:$[1],1:) (ReturnType=IEC_USINT, ArgType1=IEC_REAL, Inline=Yes)
    LREAL_TO_USINT = ToUInt(:$[1],1:) (ReturnType=IEC_USINT, ArgType1=IEC_LREAL, Inline=Yes)
    BOOL_TO_SINT = ToInt(:$[1],1:) (ReturnType=IEC_SINT, ArgType1=IEC_BOOL, Inline=Yes)
    USINT_TO_SINT = ToInt(:$[1],1:) (ReturnType=IEC_SINT, ArgType1=IEC_USINT, Inline=Yes)
    UINT_TO_SINT = ToInt(:$[1],1:) (ReturnType=IEC_SINT, ArgType1=IEC_UINT, Inline=Yes)
    INT_TO_SINT = ToInt(:$[1],1:) (ReturnType=IEC_SINT, ArgType1=IEC_INT, Inline=Yes)
    UDINT_TO_SINT = ToInt(:$[1],1:) (ReturnType=IEC_SINT, ArgType1=IEC_UDINT, Inline=Yes)
    DINT_TO_SINT = ToInt(:$[1],1:) (ReturnType=IEC_SINT, ArgType1=IEC_DINT, Inline=Yes)
    REAL_TO_SINT = ToInt(:$[1],1:) (ReturnType=IEC_SINT, ArgType1=IEC_REAL, Inline=Yes)
    LREAL_TO_SINT = ToInt(:$[1],1:) (ReturnType=IEC_SINT, ArgType1=IEC_LREAL, Inline=Yes)
    BOOL_TO_UINT = ToUInt(:$[1],2:) (ReturnType=IEC_UINT, ArgType1=IEC_BOOL, Inline=Yes)
    SINT_TO_UINT = ToUInt(:$[1],2:) (ReturnType=IEC_UINT, ArgType1=IEC_SINT, Inline=Yes)
    USINT_TO_UINT = ToUInt(:$[1],2:) (ReturnType=IEC_UINT, ArgType1=IEC_USINT, Inline=Yes)
    INT_TO_UINT = ToUInt(:$[1],2:) (ReturnType=IEC_UINT, ArgType1=IEC_INT, Inline=Yes)
    UDINT_TO_UINT = ToUInt(:$[1],2:) (ReturnType=IEC_UINT, ArgType1=IEC_UDINT, Inline=Yes)
    DINT_TO_UINT = ToUInt(:$[1],2:) (ReturnType=IEC_UINT, ArgType1=IEC_DINT, Inline=Yes)
    REAL_TO_UINT = ToUInt(:$[1],2:) (ReturnType=IEC_UINT, ArgType1=IEC_REAL, Inline=Yes)
    LREAL_TO_UINT = ToUInt(:$[1],2:) (ReturnType=IEC_UINT, ArgType1=IEC_LREAL, Inline=Yes)
    BOOL_TO_INT = ToInt(:$[1],2:) (ReturnType=IEC_INT, ArgType1=IEC_BOOL, Inline=Yes)
    SINT_TO_INT = ToInt(:$[1],2:) (ReturnType=IEC_INT, ArgType1=IEC_SINT, Inline=Yes)
    USINT_TO_INT = ToInt(:$[1],2:) (ReturnType=IEC_INT, ArgType1=IEC_USINT, Inline=Yes)
    UINT_TO_INT = ToInt(:$[1],2:) (ReturnType=IEC_INT, ArgType1=IEC_UINT, Inline=Yes)
    UDINT_TO_INT = ToInt(:$[1],2:) (ReturnType=IEC_INT, ArgType1=IEC_UDINT, Inline=Yes)
    DINT_TO_INT = ToInt(:$[1],2:) (ReturnType=IEC_INT, ArgType1=IEC_DINT, Inline=Yes)
    REAL_TO_INT = ToInt(:$[1],2:) (ReturnType=IEC_INT, ArgType1=IEC_REAL, Inline=Yes)
    LREAL_TO_INT = ToInt(:$[1],2:) (ReturnType=IEC_INT, ArgType1=IEC_LREAL, Inline=Yes)
    BOOL_TO_UDINT = ToUInt(:$[1]:) (ReturnType=IEC_UDINT, ArgType1=IEC_BOOL, Inline=Yes)
    USINT_TO_UDINT = ToUInt(:$[1]:) (ReturnType=IEC_UDINT, ArgType1=IEC_USINT, Inline=Yes)
    SINT_TO_UDINT = ToUInt(:$[1]:) (ReturnType=IEC_UDINT, ArgType1=IEC_SINT, Inline=Yes)
    UINT_TO_UDINT = ToUInt(:$[1]:) (ReturnType=IEC_UDINT, ArgType1=IEC_UINT, Inline=Yes)
    INT_TO_UDINT = ToUInt(:$[1]:) (ReturnType=IEC_UDINT, ArgType1=IEC_INT, Inline=Yes)
    DINT_TO_UDINT = ToUInt(:$[1]:) (ReturnType=IEC_UDINT, ArgType1=IEC_DINT, Inline=Yes)
    REAL_TO_UDINT = ToUInt(:$[1]:) (ReturnType=IEC_UDINT, ArgType1=IEC_REAL, Inline=Yes)
    LREAL_TO_UDINT = ToUInt(:$[1]:) (ReturnType=IEC_UDINT, ArgType1=IEC_LREAL, Inline=Yes)
    TIME_TO_UDINT = ToUInt(:$[1]:) (ReturnType=IEC_UDINT, ArgType1=IEC_TIME, Inline=Yes)
    DT_TO_UDINT = ToUInt(:$[1]:) (ReturnType=IEC_UDINT, ArgType1=IEC_DT, Inline=Yes)
    BOOL_TO_DINT = ToInt(:$[1]:) (ReturnType=IEC_DINT, ArgType1=IEC_BOOL, Inline=Yes)
    USINT_TO_DINT = ToInt(:$[1]:) (ReturnType=IEC_DINT, ArgType1=IEC_USINT, Inline=Yes)
    SINT_TO_DINT = ToInt(:$[1]:) (ReturnType=IEC_DINT, ArgType1=IEC_SINT, Inline=Yes)
    UINT_TO_DINT = ToInt(:$[1]:) (ReturnType=IEC_DINT, ArgType1=IEC_UINT, Inline=Yes)
    INT_TO_DINT = ToInt(:$[1]:) (ReturnType=IEC_DINT, ArgType1=IEC_INT, Inline=Yes)
    UDINT_TO_DINT = ToInt(:$[1]:) (ReturnType=IEC_DINT, ArgType1=IEC_UDINT, Inline=Yes)
    REAL_TO_DINT = ToInt(:$[1]:) (ReturnType=IEC_DINT, ArgType1=IEC_REAL, Inline=Yes)
    LREAL_TO_DINT = ToInt(:$[1]:) (ReturnType=IEC_DINT, ArgType1=IEC_LREAL, Inline=Yes)
    TIME_TO_DINT = ToInt(:$[1]:) (ReturnType=IEC_DINT, ArgType1=IEC_TIME, Inline=Yes)
    DT_TO_DINT = ToInt(:$[1]:) (ReturnType=IEC_DINT, ArgType1=IEC_DT, Inline=Yes)
    BOOL_TO_TIME = ToTime(:$[1]:) (ReturnType=IEC_TIME, ArgType1=IEC_BOOL, Inline=Yes)
    DINT_TO_TIME = ToTime(:$[1]:) (ReturnType=IEC_TIME, ArgType1=IEC_DINT, Inline=Yes)
    UDINT_TO_TIME = ToTime(:$[1]:) (ReturnType=IEC_TIME, ArgType1=IEC_UDINT, Inline=Yes)
    BOOL_TO_DT = ToDT(:$[1]:) (ReturnType=IEC_DT, ArgType1=IEC_BOOL, Inline=Yes)
    DINT_TO_DT = ToDT(:$[1]:) (ReturnType=IEC_DT, ArgType1=IEC_DINT, Inline=Yes)
    UDINT_TO_DT = ToDT(:$[1]:) (ReturnType=IEC_DT, ArgType1=IEC_UDINT, Inline=Yes)
    BOOL_TO_REAL = ToFloat(:$[1]:) (ReturnType=IEC_REAL, ArgType1=IEC_BOOL, Inline=Yes)
    USINT_TO_REAL = ToFloat(:$[1]:) (ReturnType=IEC_REAL, ArgType1=IEC_USINT, Inline=Yes)
    SINT_TO_REAL = ToFloat(:$[1]:) (ReturnType=IEC_REAL, ArgType1=IEC_SINT, Inline=Yes)
    UINT_TO_REAL = ToFloat(:$[1]:) (ReturnType=IEC_REAL, ArgType1=IEC_UINT, Inline=Yes)
    INT_TO_REAL = ToFloat(:$[1]:) (ReturnType=IEC_REAL, ArgType1=IEC_INT, Inline=Yes)
    UDINT_TO_REAL = ToFloat(:$[1]:) (ReturnType=IEC_REAL, ArgType1=IEC_UDINT, Inline=Yes)
    DINT_TO_REAL = ToFloat(:$[1]:) (ReturnType=IEC_REAL, ArgType1=IEC_DINT, Inline=Yes)
    LREAL_TO_REAL = ToFloat(:$[1]:) (ReturnType=IEC_REAL, ArgType1=IEC_LREAL, Inline=Yes)
    TIME_TO_REAL = ToFloat(:$[1]:) (ReturnType=IEC_REAL, ArgType1=IEC_TIME, Inline=Yes)
    BOOL_TO_LREAL = ToLReal(:$[1]:) (ReturnType=IEC_LREAL, ArgType1=IEC_BOOL, Inline=Yes)
    USINT_TO_LREAL = ToLReal(:$[1]:) (ReturnType=IEC_LREAL, ArgType1=IEC_USINT, Inline=Yes)
    SINT_TO_LREAL = ToLReal(:$[1]:) (ReturnType=IEC_LREAL, ArgType1=IEC_SINT, Inline=Yes)
    UINT_TO_LREAL = ToLReal(:$[1]:) (ReturnType=IEC_LREAL, ArgType1=IEC_UINT, Inline=Yes)
    INT_TO_LREAL = ToLReal(:$[1]:) (ReturnType=IEC_LREAL, ArgType1=IEC_INT, Inline=Yes)
    UDINT_TO_LREAL = ToLReal(:$[1]:) (ReturnType=IEC_LREAL, ArgType1=IEC_UDINT, Inline=Yes)
    DINT_TO_LREAL = ToLReal(:$[1]:) (ReturnType=IEC_LREAL, ArgType1=IEC_DINT, Inline=Yes)
    REAL_TO_LREAL = ToLReal(:$[1]:) (ReturnType=IEC_LREAL, ArgType1=IEC_REAL, Inline=Yes)
    TIME_TO_LREAL = ToLReal(:$[1]:) (ReturnType=IEC_LREAL, ArgType1=IEC_TIME, Inline=Yes)
    BOOL_TO_STRING = ToString(:ToBool(:$[1]:):) (ReturnType=IEC_STRING, ArgType1=IEC_BOOL, Inline=Yes)
    USINT_TO_STRING = ToString(:ToUInt(:$[1],1:):) (ReturnType=IEC_STRING, ArgType1=IEC_USINT, Inline=Yes)
    SINT_TO_STRING = ToString(:ToInt(:$[1],1:):) (ReturnType=IEC_STRING, ArgType1=IEC_SINT, Inline=Yes)
    UINT_TO_STRING = ToString(:ToUInt(:$[1],2:):) (ReturnType=IEC_STRING, ArgType1=IEC_UINT, Inline=Yes)
    INT_TO_STRING = ToString(:ToInt(:$[1],2:):) (ReturnType=IEC_STRING, ArgType1=IEC_INT, Inline=Yes)
    UDINT_TO_STRING = ToString(:ToUInt(:$[1]:):) (ReturnType=IEC_STRING, ArgType1=IEC_UDINT, Inline=Yes)
    DINT_TO_STRING = ToString(:ToInt(:$[1]:):) (ReturnType=IEC_STRING, ArgType1=IEC_DINT, Inline=Yes)
    REAL_TO_STRING = ToString(:ToFloat(:$[1]:):) (ReturnType=IEC_STRING, ArgType1=IEC_REAL, Inline=Yes)
    LREAL_TO_STRING = ToString(:ToLReal(:$[1]:):) (ReturnType=IEC_STRING, ArgType1=IEC_LREAL, Inline=Yes)
    STRING_TO_BOOL = ToBool(:StrToInt(:$[1]:):) (ReturnType=IEC_BOOL, ArgType1=IEC_STRING, Inline=Yes)
    STRING_TO_USINT = ToUInt(:StrToInt(:$[1]:),1:) (ReturnType=IEC_USINT, ArgType1=IEC_STRING, Inline=Yes)
    STRING_TO_SINT = ToInt(:StrToInt(:$[1]:),1:) (ReturnType=IEC_SINT, ArgType1=IEC_STRING, Inline=Yes)
    STRING_TO_UINT = ToUInt(:StrToInt(:$[1]:),2:) (ReturnType=IEC_UINT, ArgType1=IEC_STRING, Inline=Yes)
    STRING_TO_INT = ToInt(:StrToInt(:$[1]:),2:) (ReturnType=IEC_INT, ArgType1=IEC_STRING, Inline=Yes)
    STRING_TO_UDINT = ToUInt(:StrToInt(:$[1]:):) (ReturnType=IEC_UDINT, ArgType1=IEC_STRING, Inline=Yes)
    STRING_TO_DINT = ToInt(:StrToInt(:$[1]:):) (ReturnType=IEC_DINT, ArgType1=IEC_STRING, Inline=Yes)
    STRING_TO_REAL = ToFloat(:ToLReal(:$[1]:):) (ReturnType=IEC_REAL, ArgType1=IEC_STRING, Inline=Yes)
    STRING_TO_LREAL = ToLReal(:$[1]:) (ReturnType=IEC_LREAL, ArgType1=IEC_STRING, Inline=Yes)
    LEN = __LEN(:$[1]:) (ReturnType=IEC_INT, ArgType1=IEC_STRING, Inline=Yes)
    LEFT = __LEFT(:$[1], $[2]:) (ReturnType=IEC_STRING, ArgType1=IEC_STRING, ArgType2=IEC_INT, Inline=Yes)
    RIGHT = __RIGHT(:$[1], $[2]:) (ReturnType=IEC_STRING, ArgType1=IEC_STRING, ArgType2=IEC_INT, Inline=Yes)
    MID = __MID(:$[1], $[2], $[3]:) (ReturnType=IEC_STRING, ArgType1=IEC_STRING, ArgType2=IEC_INT, ArgType3=IEC_INT, Inline=Yes)
    CONCAT = __CONCAT(:$[1], $[2]:) (ReturnType=IEC_STRING, ArgType1=IEC_STRING, ArgType2=IEC_STRING, Inline=Yes)
    INSERT = __INSERT(:$[1], $[2], $[3]:) (ReturnType=IEC_STRING, ArgType1=IEC_STRING, ArgType2=IEC_STRING, ArgType3=IEC_INT, Inline=Yes)
    DELETE = __DELETE(:$[1], $[2], $[3]:) (ReturnType=IEC_STRING, ArgType1=IEC_STRING, ArgType2=IEC_INT, ArgType3=IEC_INT, Inline=Yes)
    REPLACE = __REPLACE(:$[1], $[2], $[3], $[4]:) (ReturnType=IEC_STRING, ArgType1=IEC_STRING, ArgType2=IEC_STRING, ArgType3=IEC_INT, ArgType4=IEC_INT, Inline=Yes)
    FIND = __FIND(:$[1], $[2]:) (ReturnType=IEC_INT, ArgType1=IEC_STRING, ArgType2=IEC_STRING, Inline=Yes)
    IP_INST_NUM = IpInstNum(::) (ReturnType=IEC_INT, NumArgs=0)
    IP_OWNER_ID = IpOwnerId(::) (ReturnType=IEC_INT, NumArgs=0)
    PACKET_DATA_ADR = GetIpInt(:6:) (ReturnType=IEC_UDINT, NumArgs=0, Inline=Yes)
    PACKET_COMMAND_ADR = GetIpInt(:7:) (ReturnType=IEC_UDINT, NumArgs=0, Inline=Yes)
  Parameters:
    QUOTED (QuotedName=$R, ValueType=FLOAT, ReturnType=IEC_LREAL)
      ARG (ref=EXPR, DataType=INT, MinValue=0, MaxValue=999)
    QUOTED (QuotedName=$P, ValueType=FLOAT, ReturnType=IEC_LREAL)
      ARG (ref=EXPR, DataType=INT, MinValue=0, MaxValue=999)
    QUOTED (QuotedName=$EXB, ValueType=INT, ReturnType=IEC_SINT)
      ARG (ref=EXPR, DataType=INT, MinValue=0, MaxValue=99)
    QUOTED (QuotedName=$EXW, ValueType=INT, ReturnType=IEC_INT)
      ARG (ref=EXPR, DataType=INT, MinValue=0, MaxValue=99)
    QUOTED (QuotedName=$EXL, ValueType=INT, ReturnType=IEC_DINT)
      ARG (ref=EXPR, DataType=INT, MinValue=0, MaxValue=99)
    QUOTED (QuotedName=$EXF, ValueType=FLOAT, ReturnType=IEC_REAL)
      ARG (ref=EXPR, DataType=INT, MinValue=0, MaxValue=3999)
    QUOTED (QuotedName=$MW, Synchronous=Yes, ValueType=INT, ReturnType=IEC_INT)
      ARG (ref=EXPR, DataType=INT, MinValue=0, MaxValue=99)
    QUOTED (QuotedName=$ML, Synchronous=Yes, ValueType=INT, ReturnType=IEC_DINT)
      ARG (ref=EXPR, DataType=INT, MinValue=0, MaxValue=99)
    QUOTED (QuotedName=$MF, Synchronous=Yes, ValueType=FLOAT, ReturnType=IEC_REAL)
      ARG (ref=EXPR, DataType=INT, MinValue=0, MaxValue=99)
  ParserData (NestedComments=No, DefaultCaseSensitive=Yes, CommentsSpanLines=Yes, ReadWholeFileBeforeParsing=Yes, ExpectMainProgStmts=No, UseFubTemplates=No, LexerType=IEC, RuntimePreventOverflow=No, RoundRealToInt=No, AllowArrayRefWithoutIndex=Yes, DeclareEnumLiteralsAsConstants=No, AllowVariableAutoDereference=Yes, AllowStructMemberAutoDereference=No, AllowPassByRefFnArgAutoReference=No, AllowNamedFnArgs=Yes, AllowUnnamedFnArgs=Yes, AllowFnArgMixedNaming=Yes, AllowFnArgsOutOfSequence=No, AllowBuiltinFnArgsOutOfSequence=Yes, AllowFnArgsOmmitted=Yes, AllowIgnoredFnReturn=Yes, AllowIgnoredExtraSubArgs=No, AllowFnStringInputArgsShort=No, RefuseBuiltinFnUnknownArgName=Yes, AllowBuiltinFnArgCaseSensitive=Yes)
    TKG_OPEN_COMMENT = (*
    TKG_CLOSE_COMMENT = *)
    TKG_IEC_LINE_COMMENT = //
    TKG_TRUE = TRUE:[^\w\d] (IsPattern=Yes)
    TKG_FALSE = FALSE:[^\w\d] (IsPattern=Yes)
    TKG_PRIM_TYPE (IsPattern=Yes)
    TKG_OPEN_BRACKET = (
    TKG_CLOSE_BRACKET = )
    TKG_OPEN_INDEXBRACKET = [
    TKG_CLOSE_INDEXBRACKET = ]
    TKG_COMMA = ,
    TKG_SUBRANGE = ..
    TKG_IEC_BINARY_INTEGER = 2#_[01][01_]+|2#[01][01_]+|2#_[01]|2#[01] (IsPattern=Yes)
    TKG_IEC_OCTAL_INTEGER = 8#_[0-7][0-7_]+|8#[0-7][0-7_]+|8#_[0-7]|8#[0-7] (IsPattern=Yes)
    TKG_IEC_HEX_INTEGER = 16#_[\da-fA-F][\da-fA-F]+|16#[\da-fA-F][\da-fA-F_]+|16#_[\da-fA-F]|16#[\da-fA-F] (IsPattern=Yes)
    TKG_REAL = \d[\d_]*\.[\d_]+[Ee][\+\-]\d[\d_]*|\d[\d_]*\.[\d_]+[Ee]\d[\d_]*|\d[\d_]*\.[\d_]+ (IsPattern=Yes)
    TKG_REAL_EXP = \d[\d_]*[Ee]\d[\d_]*|\d[\d_]*[Ee][\+\-]\d[\d_]* (IsPattern=Yes)
    TKG_INTEGER = \d|\d[\d_]+ (IsPattern=Yes)
    TKG_DOT = .
    TKG_PATHSYNCH_REC_IEC = DO_PATH_SYNCH:[^\w\d] (IsPattern=Yes, EndRuleToken=Yes)
    TKG_PATHSYNCH_END = END_PATH_SYNCH:[^\w\d] (IsPattern=Yes, EndRuleToken=Yes)
    TKG_PATHSYNCH_IPEVAL = IP_EVAL:[^\w\d] (IsPattern=Yes)
    TKG_CYCLIC_PATHSYNCH_BLOCKING_IEC = CYCLIC_PS_BL:[^\w\d] (IsPattern=Yes, EndRuleToken=Yes)
    TKG_CYCLIC_PATHSYNCH_IEC = CYCLIC_PS:[^\w\d] (IsPattern=Yes, EndRuleToken=Yes)
    TKG_CYCLIC_BLOCKING_IEC = CYCLIC_BL:[^\w\d] (IsPattern=Yes, EndRuleToken=Yes)
    TKG_CYCLIC_IEC = CYCLIC:[^\w\d] (IsPattern=Yes, EndRuleToken=Yes)
    TKG_CYCLIC_END_IEC = END_CYCLIC:[^\w\d] (IsPattern=Yes, EndRuleToken=Yes)
    TKG_REFERENCE = REFERENCE:[^\w\d] (FollowedBy=TKG_IEC_TO, IsPattern=Yes)
    TKG_IEC_TO = TO:[^\w\d] (IsPattern=Yes)
    TKG_IEC_DO = DO:[^\w\d] (IsPattern=Yes, EndRuleToken=Yes)
    TKG_FOR_NOFINALDEC = FOR:[^\w\d] (FileXLInvalid=Yes, IsPattern=Yes)
    TKG_FORSTEP = BY:[^\w\d] (FileXLInvalid=Yes, IsPattern=Yes)
    TKG_ENDFOR = END_FOR:[^\w\d] (FileXLInvalid=Yes, IsPattern=Yes, EndRuleToken=Yes)
    TKG_IF = IF:[^\w\d] (IsPattern=Yes)
    TKG_THEN = THEN:[^\w\d] (IsPattern=Yes, EndRuleToken=Yes)
    TKG_BLOCK_ELSEIF = ELSIF:[^\w\d] (IsPattern=Yes)
    TKG_ELSE_AND_DEFAULT = ELSE:[^\w\d] (IsPattern=Yes, EndRuleToken=Yes)
    TKG_BLOCK_ENDIF = END_IF:[^\w\d] (IsPattern=Yes, EndRuleToken=Yes)
    TKG_SWITCH = CASE:[^\w\d] (IsPattern=Yes, FileXLInvalid=Yes)
    TKG_ENDSWITCH_NOBREAK = END_CASE:[^\w\d] (FileXLInvalid=Yes, IsPattern=Yes, EndRuleToken=Yes)
    TKG_WHILE = WHILE:[^\w\d] (FileXLInvalid=Yes, IsPattern=Yes)
    TKG_ENDWHILE = END_WHILE:[^\w\d] (FileXLInvalid=Yes, IsPattern=Yes, EndRuleToken=Yes)
    TKG_DO = REPEAT:[^\w\d] (FileXLInvalid=Yes, IsPattern=Yes, EndRuleToken=Yes)
    TKG_ENDDO_UNTIL = UNTIL:[^\w\d] (FileXLInvalid=Yes, IsPattern=Yes)
    TKG_ENDDO_POSTCOND = END_REPEAT:[^\w\d] (FileXLInvalid=Yes, IsPattern=Yes, EndRuleToken=Yes)
    TKG_BREAK = EXIT:[^\w\d] (FileXLInvalid=Yes, IsPattern=Yes)
    TKG_RETURN = RETURN:[^\w\d] (FileXLInvalid=Yes, IsPattern=Yes)
    TKG_IEC_SEL_FN = SEL:[^\w\d] (FileXLInvalid=Yes, IsPattern=Yes)
    TKG_IEC_MUX_FN = MUX:[^\w\d] (FileXLInvalid=Yes, IsPattern=Yes)
    TKG_TIME_LITERAL = time#\-[dDhHmMsS_\.\d]+|time#[dDhHmMsS_\.\d]+|t#\-[dDhHmMsS_\.\d]+|t#[dDhHmMsS_\.\d]+ (CaseSensitive=no, IsPattern=yes)
    TKG_DATE_AND_TIME_LITERAL = DT#[12]\d\d\d\-[\d\:\-]*|DATE_AND_TIME#[12]\d\d\d\-[\d\:\-]* (CaseSensitive=no, IsPattern=yes)
    TKG_DATE_LITERAL = D#[12]\d\d\d\-[\d\-]*|DATE#[12]\d\d\d\-[\d\-]* (CaseSensitive=no, IsPattern=yes)
    TKG_TIME_OF_DAY_LITERAL = TOD#\d[\d\:\.]*|TIME_OF_DAY#\d[\d\:\.]* (CaseSensitive=no, IsPattern=yes)
    TKG_ASSIGN_EQ = :=
    TKG_OPEN_IP_EXTENSION = {
    TKG_CLOSE_IP_EXTENSION = }
    TKG_IEC_OPEN_TYPE = TYPE:[^\w\d] (IsPattern=Yes)
    TKG_IEC_CLOSE_TYPE = END_TYPE:[^\w\d] (IsPattern=Yes, EndRuleToken=Yes)
    TKG_VAR = VAR:[^\w\d] (IsPattern=Yes)
    TKG_VAR_GLOBAL = VAR_GLOBAL:[^\w\d] (IsPattern=Yes)
    TKG_VAR_INPUT = VAR_INPUT:[^\w\d] (IsPattern=Yes)
    TKG_VAR_OUTPUT = VAR_OUTPUT:[^\w\d] (IsPattern=Yes)
    TKG_VAR_IN_OUT = VAR_IN_OUT:[^\w\d] (IsPattern=Yes)
    TKG_VAR_END = END_VAR:[^\w\d] (IsPattern=Yes, EndRuleToken=Yes)
    TKG_VAR_RETAIN = RETAIN:[^\d\w] (IsPattern=Yes)
    TKG_IP_RETAIN = IP_RETAIN:[^\d\w] (IsPattern=Yes)
    TKG_AT = AT:[^\d\w] (IsPattern=Yes)
    TKG_PLC = PLC:[^\d\w] (IsPattern=Yes)
    TKG_PV_UNDECL = UNRETAIN_VAR:[^\d\w] (IsPattern=Yes)
    TKG_VARSYNCH_IP = IP_SYNCH:[^\d\w] (IsPattern=Yes)
    TKG_VARSYNCH_PATH = PATH_SYNCH:[^\d\w] (IsPattern=Yes)
    TKG_CONSTANT = CONSTANT:[^\d\w] (IsPattern=Yes)
    TKG_VARSCOPE_IP_GLOBAL = IP_GLOBAL:[^\w\d] (IsPattern=Yes)
    TKG_VARSCOPE_SHARED_IP_GLOBAL = SHARED_IP_GLOBAL:[^\w\d] (IsPattern=Yes)
    TKG_VARSCOPE_NC_GLOBAL = NC_GLOBAL:[^\w\d] (IsPattern=Yes)
    TKG_VARSCOPE_PLC_GLOBAL = PLC_GLOBAL:[^\w\d] (IsPattern=Yes)
    TKG_VARSCOPE_IP_LOCAL = LOCAL:[^\w\d] (IsPattern=Yes)
    TKG_IEC_NAMESPACE_SPEC = :: (IsPattern=No)
    TKG_IEC_DATATYPE_SPEC = : (IsPattern=No)
    TKG_IEC_ARRAY = ARRAY:[^\w\d] (IsPattern=Yes)
    TKG_IEC_OF = OF:[^\w\d] (IsPattern=Yes)
    TKG_IEC_DELIM = ; (EndRuleToken=Yes)
    TKG_IEC_OPEN_STRUCT = STRUCT:[^\w\d] (IsPattern=Yes)
    TKG_IEC_CLOSE_STRUCT = END_STRUCT:[^\w\d] (IsPattern=Yes)
    TKG_BITWISE_LP_BINARY_AND = AND:[^\w\d] (IsPattern=Yes)
    TKG_BITWISE_LP_BINARY_OR = OR:[^\w\d] (IsPattern=Yes)
    TKG_BITWISE_LP_BINARY_XOR = XOR:[^\w\d] (IsPattern=Yes)
    TKG_BITWISE_UNARY_COMPLEMENT = NOT:[^\w\d] (IsPattern=Yes)
    TKG_COMP_EXACT_BINARY_GREATER_THAN_OR_EQ = >=
    TKG_COMP_EXACT_BINARY_LESS_THAN_OR_EQ = <=
    TKG_COMP_EXACT_BINARY_EQUAL_TO = =
    TKG_COMP_EXACT_BINARY_NOT_EQUAL_TO = <>
    TKG_COMP_EXACT_BINARY_GREATER_THAN = >
    TKG_COMP_EXACT_BINARY_LESS_THAN = <
    TKG_ARITH_BINARY_PLUS = +
    TKG_ARITH_BINARY_MINUS = -
    TKG_ARITH_BINARY_POWER = **
    TKG_ARITH_BINARY_MULTIPLY = *
    TKG_ARITH_BINARY_DIVIDE = /
    TKG_ARITH_BINARY_MODULO = MOD:[^\w\d] (IsPattern=Yes)
    TKG_PRAGMA = #pragma:[^\w\d] (IsPattern=Yes, FollowedBy=TKG_IDENTIFIER)
    TKG_INCLUDE = #include:[^\w\d] (IsPattern=Yes)
    TKG_PROG_START = PROGRAM:[^\w\d] (IsPattern=Yes, FollowedBy=TKG_PROG_NAME)
    TKG_PROG_NAME = _INIT:[^\w\d]|_CYCLIC:[^\w\d]|_EXIT:[^\w\d]|_MAIN:[^\w\d] (IsPattern=Yes, EndRuleToken=Yes)
    TKG_PROG_END = END_PROGRAM:[^\w\d] (IsPattern=Yes, EndRuleToken=Yes)
    TKG_SUBPROG_START = FUNCTION:[^\w\d] (IsPattern=Yes)
    TKG_SUBPROG_END = END_FUNCTION:[^\w\d] (IsPattern=Yes, EndRuleToken=Yes)
    TKG_FUB_DECL = FUNCTION_BLOCK:[^\w\d] (IsPattern=Yes)
    TKG_FUB_END = END_FUNCTION_BLOCK:[^\w\d] (IsPattern=Yes, EndRuleToken=Yes)
    TKG_RETURN = RETURN:[^\w\d] (IsPattern=Yes)
    TKG_ACCESS = ACCESS:[^\w\d] (IsPattern=Yes)
    TKG_DEREF_OP = ^
    TKG_ACTION = ACTION:[^\w\d] (IsPattern=Yes)
    TKG_ACTION_END = END_ACTION:[^\w\d] (IsPattern=Yes, EndRuleToken=Yes)
    TKG_IEC_TYPED_VALUE = \w#:[\w\d\+\-]|\w[\w\d]+#:[\w\d\+\-] (IsPattern=Yes)
    TKG_PARAM_PREFIX = $R:[^\w\d]|$P:[^\w\d]|$MW:[^\w\d]|$ML:[^\w\d]|$MF:[^\w\d]|$EXW:[^\w\d]|$EXL:[^\w\d]|$EXF:[^\w\d]|$EXB:[^\w\d] (IsPattern=Yes)
    TKG_IDENTIFIER = \w|\w[\w\d$]+|$[\w\d$]+ (IsPattern=Yes)
    TKG_INIT_IDENTIFIER = \w|\w[\w\d$]+|$[\w\d$]+ (IsPattern=Yes, Disabled=Yes)
  StringChars (AsciiStringStart=', AsciiStringEnd=', UTF16StringStart=", UTF16StringEnd=")
    EscapeSeq (Search=$N, CaseSensitive=Yes, ReplaceValue=10)
    EscapeSeq (Search=$n, CaseSensitive=Yes, ReplaceValue=10)
    EscapeSeq (Search=$L, CaseSensitive=Yes, ReplaceValue=10)
    EscapeSeq (Search=$l, CaseSensitive=Yes, ReplaceValue=10)
    EscapeSeq (Search=$P, CaseSensitive=Yes, ReplaceValue=12)
    EscapeSeq (Search=$p, CaseSensitive=Yes, ReplaceValue=12)
    EscapeSeq (Search=$R, CaseSensitive=Yes, ReplaceValue=13)
    EscapeSeq (Search=$r, CaseSensitive=Yes, ReplaceValue=13)
    EscapeSeq (Search=$T, CaseSensitive=Yes, ReplaceValue=9)
    EscapeSeq (Search=$t, CaseSensitive=Yes, ReplaceValue=9)
    EscapeSeq (Search=$', CaseSensitive=Yes, ReplaceStr=')
    EscapeSeq (Search=$", CaseSensitive=Yes, ReplaceStr=")
    EscapeSeq (Search=$[\dA-Fa-f]+, IsPattern=Yes, CaseSensitive=Yes, ReplaceEncodingBase=16)
    EscapeSeq (Search=$$, ReplaceStr=$)
    EscapeSeq (Search=$, ReplaceStr=)
```

- Data object Logical/GmcIpConfig/gmciplbr (Cnc, version 3.13.0) (no source held here)

- Data object Logical/GmcIpConfig/gmciplog (Cnc, version 3.13.0) (no source held here)

### Data object Logical/GmcIpConfig/gmciplsm (Cnc, version 3.13.0)

#### gmciplsm.cnc
```
Root (LangModule=ailgcode, Version=1.0)
  PrimTypes (CaseSensitive=No)
    REAL (BRType=LREAL)
    INT (BRType=DINT)
    CHAR (BRType=USINT)
    BOOL (BRType=BOOL)
    STRING (BRType=STRING)
    AXIS (BRType=AXIS)
    BR_LREAL (BRType=LREAL)
    BR_REAL (BRType=REAL)
    BR_UDINT (BRType=UDINT)
    BR_DINT (BRType=DINT)
    BR_UINT (BRType=UINT)
    BR_INT (BRType=INT)
    BR_USINT (BRType=USINT)
    BR_SINT (BRType=SINT)
    BR_BOOL (BRType=BOOL)
    BR_TIME (BRType=TIME)
    BR_DATE_AND_TIME (BRType=DATE_AND_TIME)
  Preprocess:
    PP_RULE_NCK (Search=NCK , Replace=nc_global )
    PP_RULE_CHAN (Search=CHAN , Replace=ip_global )
    PP_RULE_FRAME_I (Search=$FRAME_I, Replace=(1,0,0,0,1,0,0,0,1,0,0,0))
    PP_RULE_FRAME_DEF (IsPattern=Yes, Search=FRAME:[^\w\d], Replace=REAL[12])
  BuiltInProcs:
    cancel = beginpathsynch
        StopCyclicGroups(:${*}:);
      endpathsynch (MinArgs=1, MaxArgs=*)
    RET = #next_motion.Command = MPCMD_SET_M_FCT;
      #next_motion.Data.I4_value = 17;
      PushPacket(::);
      ReturnTo(:${*}:); (MinArgs=0, MaxArgs=4, Eval=Early, Inline=Yes)
  BuiltInFns:
    ABS = Abs(:$[1]:) (NumArgs=1, Inline=Yes)
    SIN = Sin(:$[1]:) (NumArgs=1, Inline=Yes)
    COS = Cos(:$[1]:) (NumArgs=1, Inline=Yes)
    TAN = Tan(:$[1]:) (NumArgs=1, Inline=Yes)
    ASIN = ASin(:$[1]:) (NumArgs=1, Inline=Yes)
    ACOS = ACos(:$[1]:) (NumArgs=1, Inline=Yes)
    ATAN = ATan(:$[1]:) (NumArgs=1, Inline=Yes)
    ATAN2 = ATan2(:$[1],$[2]:) (NumArgs=2, Inline=Yes)
    SQRT = Sqrt(:$[1]:) (NumArgs=1, Inline=Yes)
    POT = (($[1])*($[1])) (NumArgs=1, Inline=Yes)
    TRUNC = Fix(:$[1]:) (NumArgs=1, Inline=Yes)
    ROUND = Round(:$[1]:) (NumArgs=1, Inline=Yes)
    LN = Ln(:$[1]:) (NumArgs=1, Inline=Yes)
    EXP = Exp(:$[1]:) (NumArgs=1, Inline=Yes)
    MINVAL = MinVal(:$[1], $[2]:) (NumArgs=2, Inline=Yes)
    MAXVAL = MaxVal(:$[1], $[2]:) (NumArgs=2, Inline=Yes)
    BOUND = Bounds(:$[1], $[2], $[3]:) (NumArgs=3, Inline=Yes)
    TO_BOOL = ToBool(:$[1]:) (NumArgs=1, Inline=Yes)
    TO_INT = ToInt(:$[1]:) (NumArgs=1, Inline=Yes)
    TO_CHAR = ToChar(:$[1]:) (NumArgs=1, Inline=Yes)
    TO_REAL = ToLReal(:$[1]:) (NumArgs=1, Inline=Yes)
    TO_FLOAT = ToFloat(:$[1]:) (NumArgs=1, Inline=Yes)
    DEFINED = Defined(:$[1]:) (NumArgs=1, Inline=Yes)
    TIME_MS = TimeMs(::) (NumArgs=0)
    SET = ${*} (MinArgs=0, MaxArgs=*, Inline=Yes)
    REP = ArrayRep(:${*}:) (MinArgs=1, MaxArgs=2, Inline=Yes)
    ADR = Adr(:\$[1]:) (NumArgs=1, Inline=Yes)
    SIZEOF = Sizeof(:\$[1]:) (NumArgs=1, Inline=Yes)
    NUM_LOADED_FILES = NumLoadedFiles(::) (NumArgs=0)
    NUM_LOADED_PROG_FILES = NumLoadedProgFiles(::) (NumArgs=0)
    MEM_SIZE_IP_ALL = MemSizeIpInstAll(::) (NumArgs=0)
    MEM_SIZE_IP_LIB = MemSizeIpInst(::) (NumArgs=0)
    MEM_SIZE_SHLIB = MemSizeShLib(::) (NumArgs=0)
    MEM_SIZE_FILE = MemSizeFile(:$[1]:) (MinArgs=0, MaxArgs=1)
    MEM_SIZE_IP_STACK_SPACE = MemStackSpace(::) (NumArgs=0)
  AxesSpec:
    AxisRef = $\s*=\s*AC (Mode=3)
    AxisRef = $\s*=\s*IC (Mode=4)
  PVMacros:
    SBLOF (ArrayDims=0, Group=500)
      CALL = #call->forbid_stepping = 1; (Inline=Yes)
    SBLON (ArrayDims=0, Group=500)
      CALL = #call->forbid_stepping = 0; (Inline=Yes)
    DISPLOF (ArrayDims=0, Group=500)
      CALL = #call->forbid_display = 1; (Inline=Yes)
    DISPLON (ArrayDims=0, Group=500)
      CALL = #call->forbid_display = 0; (Inline=Yes)
    RDISABLE (ArrayDims=0, Group=500)
      CALL = @#job->sa.keep_alive = 1;
        @#thread.sa_keep_alive = 1; (Inline=Yes)
    P_SUBPAR $P_SUBPAR (ArrayDims=1, Group=500)
      GET = return ArgNumIsDefined(:$[1]:);
    P_STACK $P_STACK:
      GET = return UserCallDepth(::);
  FubTemplates:
    StdFubTemplate (IsDefault=Yes, Inline=Yes)
      Arg (ref=FUBINST, DataType=FLOAT)
      Arg (ref=FUBERRLEV, DataType=FLOAT)
      Arg (ref=PATHSYNCH, DataType=FLOAT)
      Arg (ref=BLOCKING, DataType=FLOAT)
  SynchActions:
    SABlocks:
      default (IsDefault=Yes)
        cyclic (Inline=Yes)
          Arg (ref=ACTIONS, DataType=STATEMENTS)
          Arg (ref=ID, DataType=FLOAT, DefaultInt=-1, MinCount=0, MaxCount=1)
      whenever:
        cyclic (Inline=Yes)
          Arg (ref=COND, DataType=FLOAT)
          Arg (ref=ACTIONS, DataType=STATEMENTS)
          Arg (ref=ID, DataType=FLOAT, DefaultInt=-1, MinCount=0, MaxCount=1)
      when:
        cyclic (Inline=Yes)
          Arg (ref=COND, DataType=FLOAT)
          Arg (ref=ACTIONS, DataType=STATEMENTS)
          Arg (ref=ID, DataType=FLOAT, DefaultInt=-1, MinCount=0, MaxCount=1)
      every:
        cyclic (Inline=Yes)
          Arg (ref=COND, DataType=FLOAT)
          Arg (ref=ACTIONS, DataType=STATEMENTS)
          Arg (ref=ID, DataType=FLOAT, DefaultInt=-1, MinCount=0, MaxCount=1)
      from:
        cyclic (Inline=Yes)
          Arg (ref=COND, DataType=FLOAT)
          Arg (ref=ACTIONS, DataType=STATEMENTS)
          Arg (ref=ID, DataType=FLOAT, DefaultInt=-1, MinCount=0, MaxCount=1)
    NonModalActivation:
      Start = @#thread.sa_last_keep_alive = 1;
        ActivateCyclicGroup(:-1:);
      Stop = WaitStopCyclicGroups(:(:-1:):);
  ParserData (NestedComments=Yes, DefaultCaseSensitive=No, CommentsSpanLines=No, SubDeclsLocalToFile=Yes, ProgDeclsLocalToFile=Yes, AllowUnprefixedFileCalls=Yes, AllowUnprefixedSubCalls=Yes, LocalVarScopeForMainProg=No, FileScopeVarsVisibleInSub=Yes, MainPrgReturnAtNextMainPrgHdr=Yes, AllowVarReadBeforeAssign=No, AllowArrayRefWithoutIndex=Yes, AllowNamedFnArgs=Yes, AllowBuiltinFnArgsOutOfSequence=Yes, AllowBuiltInProcCallWithoutBrackets=Yes, AllowBuiltInFnCallWithoutBrackets=No, AllowPLCFnCallWithoutBrackets=No, AllowStructMemberAutoDereference=Yes, AllowVariableAutoDereference=Yes, EnableStringCharacterIndexing=Yes, AllowIgnoredExtraSubArgs=Yes, OnMacroRedefinition=Error, CheckFileTimestampBeforeCalls=Yes)
    TKG_END_OF_LINE = \n (IsPattern=No)
    TKG_LINE_CONTINUE = \ (IsPattern=No, FileXLInvalid=Yes)
    TKG_LINE_BREAK = @@
    TKG_OPEN_COMMENT = ;
    TKG_CLOSE_COMMENT
    TKG_TRUE = TRUE:\W (IsPattern=Yes)
    TKG_FALSE = FALSE:\W (IsPattern=Yes)
    TKG_PAREVAL_MODAL_ID = ID:[\s=] (FileXLInvalid=Yes, IsPattern=Yes)
    TKG_MACRO_DEFINE_GLOBAL = define\s+ip_global:\s (IsPattern=Yes, FollowedBy=TKG_MACRO_NAME)
    TKG_MACRO_DEFINE = define\s+local:\s|define:\s (IsPattern=Yes, FollowedBy=TKG_MACRO_NAME)
    TKG_MACRO_UNDEFINE = undefine:\s (IsPattern=Yes, FollowedBy=TKG_MACRO_NAME)
    TKG_MACRO_AS = as:[\s\n] (IsPattern=Yes, FollowedBy=TKG_MACRO_TEXT)
    TKG_PROG_START = %:[^L] (IsPattern=Yes, CaseSensitive=Yes, FollowedBy=TKG_PROG_NAME)
    TKG_PROG_NAME = [\w\d]+ (IsPattern=Yes, Restricted=Yes)
    TKG_SET_MODAL_SUB = MCALL:\W (FileXLInvalid=Yes, IsPattern=Yes)
    TKG_INDIR_PROG_CALL = CALL:\s (IsPattern=Yes)
    TKG_INDIR_PROG_BLOCK = BLOCK:\s (FileXLInvalid=Yes, IsPattern=Yes)
    TKG_PROC_START = PROC:\s (FileXLInvalid=Yes, IsPattern=Yes, FollowedBy=TKG_PROC_NAME)
    TKG_PROC_NAME = \w[\w\d]+ (IsPattern=Yes, Restricted=Yes)
    TKG_ARG_PASSBYREF = VAR:\s (IsPattern=Yes)
    TKG_SUBPROG_PROTO = INTERN:\s (IsPattern=Yes, FollowedBy=TKG_SUBPROG_NAME)
    TKG_SUBPROG_START = SUB\s|%:L (FileXLInvalid=Yes, IsPattern=Yes, CaseSensitive=Yes, FollowedBy=TKG_SUBPROG_NAME)
    TKG_SUBPROG_NAME = \w[\w\d]+ (IsPattern=Yes, Restricted=Yes)
    TKG_EXTERN = EXTERN:\s (IsPattern=Yes, FollowedBy=TKG_PROG_FILE_NAME)
    TKG_PROG_FILE_NAME = [\^#&@']?[\w\d\./\:]+ (IsPattern=Yes, Restricted=Yes)
    TKG_PV_DECL = def:\s (IsPattern=Yes)
    TKG_PV_UNDECL = ~def:\s (IsPattern=Yes)
    TKG_VAR_RETAIN = retain:\s (IsPattern=Yes)
    TKG_VARSCOPE_IP_LOCAL = local:[\s\n] (IsPattern=Yes)
    TKG_VARSCOPE_IP_GLOBAL = ip_global:[\s\n] (IsPattern=Yes)
    TKG_VARSCOPE_NC_GLOBAL = nc_global:[\s\n] (IsPattern=Yes)
    TKG_VARSCOPE_PLC_GLOBAL = plc_global:[\s\n] (IsPattern=Yes)
    TKG_VARSYNCH_IP = ip_synch:\s (IsPattern=Yes)
    TKG_VARSYNCH_PATH = path_synch:\s (IsPattern=Yes)
    TKG_PAREVAL_DO = do:\s (FileXLInvalid=Yes, IsPattern=Yes)
    TKG_GOTOF = gotof:\s (FileXLInvalid=Yes, IsPattern=Yes, OptFollowedBy=TKG_GOTO_DEST)
    TKG_GOTOB = gotob:\s (FileXLInvalid=Yes, IsPattern=Yes, OptFollowedBy=TKG_GOTO_DEST)
    TKG_GOTO = goto:\s (FileXLInvalid=Yes, IsPattern=Yes, OptFollowedBy=TKG_GOTO_DEST)
    TKG_GOTO_DEST = \w[\w\d]* (IsPattern=Yes, Restricted=Yes)
    TKG_ARITH_BINARY_INT_DIVIDE = DIV:[\s(] (IsPattern=Yes)
    TKG_ARITH_BINARY_MODULO = MOD:[\s(] (IsPattern=Yes)
    TKG_FOR = FOR:\s (FileXLInvalid=Yes, IsPattern=Yes)
    TKG_ENDFOR = ENDFOR:[\s\n] (FileXLInvalid=Yes, IsPattern=Yes)
    TKG_FORTO = TO:\W (IsPattern=Yes)
    TKG_DO = repeat:[\s\n] (FileXLInvalid=Yes, IsPattern=Yes)
    TKG_ENDDO_UNTIL = until:[\s(] (FileXLInvalid=Yes, IsPattern=Yes)
    TKG_LOGICAL_UNARY_NOT = not:\W (IsPattern=Yes)
    TKG_SUPPRESS_SINGLE_STEP = NOHALT
    TKG_NC_BLOCK_PREFIX = N:[\s\d] (IsPattern=Yes)
    TKG_LOGICAL_HP_BINARY_AND = and:\W (IsPattern=Yes)
    TKG_LOGICAL_HP_BINARY_OR = or:\W (IsPattern=Yes)
    TKG_LOGICAL_HP_BINARY_XOR = xor:\W (IsPattern=Yes)
    TKG_BITWISE_BINARY_AND = b_and:\W (IsPattern=Yes)
    TKG_BITWISE_BINARY_OR = b_or:\W (IsPattern=Yes)
    TKG_BITWISE_BINARY_XOR = b_xor:\W (IsPattern=Yes)
    TKG_BITWISE_UNARY_COMPLEMENT = b_not:\W (IsPattern=Yes)
    TKG_IF = if:\W (FileXLInvalid=Yes, IsPattern=Yes)
    TKG_THEN = then:\W (FileXLInvalid=Yes, IsPattern=Yes)
    TKG_BLOCK_ELSE = else:\W (FileXLInvalid=Yes, IsPattern=Yes)
    TKG_BLOCK_ENDIF = endif:\W (FileXLInvalid=Yes, IsPattern=Yes)
    TKG_SWITCH = case:\W (FileXLInvalid=Yes, IsPattern=Yes)
    TKG_SWITCH_OF = of:\W (FileXLInvalid=Yes, IsPattern=Yes)
    TKG_SWITCH_DEFAULT = default:\W (FileXLInvalid=Yes, IsPattern=Yes)
    TKG_WHILE = while:\W (FileXLInvalid=Yes, IsPattern=Yes)
    TKG_ENDWHILE = endwhile (FileXLInvalid=Yes)
    TKG_FOREVER = loop:\W (FileXLInvalid=Yes, IsPattern=Yes)
    TKG_ENDFOREVER = endloop:\W (FileXLInvalid=Yes, IsPattern=Yes)
    TKG_LABEL_DEF = \w:\:|\w[\w\d]+:\: (IsPattern=Yes, FollowedBy=TKG_LABEL_SUFFIX)
    TKG_LABEL_SUFFIX = : (Restricted=Yes)
    TKG_MACRO_TEXT = . (Restricted=Yes, IsPattern=Yes)
    TKG_MACRO_NAME = [$\w][$\w\d(]+ (Restricted=Yes, IsPattern=Yes)
    TKG_PRIM_TYPE (IsPattern=Yes)
    TKG_OPEN_BRACKET = (
    TKG_CLOSE_BRACKET = )
    TKG_OPEN_INDEXBRACKET = [
    TKG_CLOSE_INDEXBRACKET = ]
    TKG_COMMA = ,
    TKG_DOT = \.:\w (IsPattern=Yes, FollowedBy=TKG_STRUCT_MEMBER_REF)
    TKG_STRUCT_MEMBER_REF = \w|\w[\w\d]+ (IsPattern=Yes, Restricted=Yes)
    TKG_PARAM_PREFIX = R:[\[\d]|$[RP]:[\[\d]|M[WLF]:[\[\d]|EX[WLBF]:[\[\d] (IsPattern=Yes)
    TKG_SUBRANGE = ..
    TKG_NUMBER = \d+\.\d+|\d+\.:[^\.] (IsPattern=Yes)
    TKG_INTEGER = \d+ (IsPattern=Yes)
    TKG_FRACTION = \.\d+ (IsPattern=Yes)
    TKG_NUMBER_EXP = EX:[\s\d\+\-\.] (IsPattern=Yes)
    TKG_STRING_CONCAT = <<
    TKG_COMP_BINARY_GREATER_THAN_OR_EQ = >=
    TKG_COMP_BINARY_LESS_THAN_OR_EQ = <=
    TKG_COMP_BINARY_EQUAL_TO = ==
    TKG_COMP_BINARY_NOT_EQUAL_TO = <>
    TKG_COMP_BINARY_GREATER_THAN = >
    TKG_COMP_BINARY_LESS_THAN = <
    TKG_ASSIGN_INCR = =ic:( (IsPattern=Yes)
    TKG_ASSIGN_EQ = =
    TKG_ARITH_BINARY_PLUS = +
    TKG_ARITH_BINARY_MINUS = -
    TKG_ARITH_BINARY_MULTIPLY = *
    TKG_ARITH_BINARY_DIVIDE = /
    TKG_SUBCALL_REPEAT_PREFIX = P:[\s\d] (IsPattern=Yes, FollowedBy=TKG_INTEGER)
    TKG_PV_DECL_REF = \w[\w\d\.\:\*]* (IsPattern=Yes, Restricted=Yes)
    TKG_G_CODE_PREFIX = G:[\s\d] (IsPattern=Yes)
    TKG_M_CODE_PREFIX = M:[\s\d(] (IsPattern=Yes)
    TKG_FUB_DECL = fub\s (IsPattern=Yes)
    TKG_FUB_ERR_LEV_1 = error_level_1:\s (IsPattern=Yes)
    TKG_FUB_ERR_LEV_2 = error_level_2:\s (IsPattern=Yes)
    TKG_FUB_ERR_LEV_3 = error_level_3:\s (IsPattern=Yes)
    TKG_FUB_ERR_LEV_4 = error_level_4:\s (IsPattern=Yes)
    TKG_FUB_BLOCKING = blocking:[\s\n] (IsPattern=Yes)
    TKG_FUB_NON_BLOCKING = non_blocking:\s (IsPattern=Yes)
    TKG_IEC_TYPED_VALUE = #[\w\d]+:[^\w\d\:] (IsPattern=Yes)
    TKG_REFERENCE = ref:[\s\n]|reference:[\s\n] (IsPattern=Yes, FollowedBy=TKG_IEC_TO)
    TKG_IEC_TO = to:[\s\n] (IsPattern=Yes, Restricted=Yes)
    TKG_ACCESS = ACCESS:[\s\n] (IsPattern=Yes)
    TKG_BINARY_LITERAL_START = 'B:[01_] (FollowedBy=TKG_BINARY_LITERAL_BODY, IsPattern=Yes)
    TKG_BINARY_LITERAL_BODY = [01_]+' (Restricted=Yes, IsPattern=Yes)
    TKG_HEX_LITERAL_START = 'H:[\dA-F_] (FollowedBy=TKG_HEX_LITERAL_BODY, IsPattern=Yes)
    TKG_HEX_LITERAL_BODY = [\dA-F_]+' (Restricted=Yes, IsPattern=Yes)
    TKG_WORD = \w|\w[\w\d\./]+|\./\w|\./\w[\w\d\./]+|[\^#][\w\d]+\:[\w\d\./]+ (IsPattern=Yes)
  StringChars (AsciiStringStart=", AsciiStringEnd=", UTF16StringStart=W", UTF16StringEnd=")
    EscapeSeq (Search=$N, ReplaceValue=10)
    EscapeSeq (Search=$L, ReplaceValue=10)
    EscapeSeq (Search=$P, ReplaceValue=12)
    EscapeSeq (Search=$R, ReplaceValue=13)
    EscapeSeq (Search=$T, ReplaceValue=9)
    EscapeSeq (Search=$Q, ReplaceStr=")
    EscapeSeq (Search=$', ReplaceStr=')
    EscapeSeq (Search=$", ReplaceStr=")
    EscapeSeq (Search=$[\dA-Fa-f]+, IsPattern=Yes, ReplaceEncodingBase=16)
    EscapeSeq (Search=$$, ReplaceStr=$)
    EscapeSeq (Search=$, ReplaceStr=)
```

- Data object Logical/GmcIpConfig/gmcipmx (Cnc, version 3.13.0) (no source held here)

### gmcipmxd.cnc
```
(********************************************************************
 * COPYRIGHT -- Bernecker + Rainer
 ********************************************************************
 * Library: Motion Command Extension
 * File: arnc0mx.typ
 * Author: B&R
 ********************************************************************
 * Data types of Motion Command Library
 ********************************************************************)

TYPE
	MXOrientationType : STRUCT
		Type : UDINT;
		Angle : ARRAY[0..3]OF LREAL;
	END_STRUCT;
	MXPositionType : STRUCT
		x : LREAL;
		y : LREAL;
		z : LREAL;
	END_STRUCT;
	MXFrameType : 	STRUCT
		Pos : MXPositionType;
		Orient : MXOrientationType;
	END_STRUCT;
	MXToolType : STRUCT
		Frame : MXFrameType;
		Radius : LREAL;
	END_STRUCT;
	MXJointAxisType :ARRAY[0..5]OF LREAL;
	MXAuxAxisType :ARRAY[0..14]OF LREAL;
	MXBaseAxisType :ARRAY[0..5]OF LREAL;
	MXRotAxisType :ARRAY[0..5]OF LREAL;
	MXConfigType : 	STRUCT
		Mode : UDINT;
	END_STRUCT;
	MXPointType : 	STRUCT
		Pos : MXPositionType;
		Orient : MXOrientationType;
		Cfg : MXConfigType;
		RotAxis : MXRotAxisType;
		AuxAxis : MXAuxAxisType;
	END_STRUCT;
	MXPathTransType : STRUCT
		Radius	:	LREAL;
		Type	:	UDINT;
	END_STRUCT;
	MXPathDescType : STRUCT
		Trans	:	MXPathTransType;
	END_STRUCT;
	MXOptMotType : STRUCT
		Enable : BOOL;
		VelPathDef : USINT;
		RobotPar : USINT;
		Limits : USINT;
	END_STRUCT;
	MXDynamicDescType :	STRUCT
		Accel : LREAL := 100;
		Decel : LREAL := 100;
		Optmot : MXOptMotType;
	END_STRUCT;
	MXHWTrigType : 	STRUCT
		Source : USINT;
		Index : USINT;
	END_STRUCT;
	MXSWTrigType : STRUCT
		Expression : STRING[64];
	END_STRUCT;
	MXTriggConfigType :	STRUCT
		Type : UINT;
		HWTrig : MXHWTrigType;
		SWTrig : MXSWTrigType;
		Edge : USINT;
		ResidPath : USINT;
	END_STRUCT;
	MXVelocityType : STRUCT
		v : LREAL;
		Mode : UDINT := 1;
	END_STRUCT;
	MXAxisTargetType : 	STRUCT
		JointAxis : MXJointAxisType;
		AuxAxis : MXAuxAxisType;
		BaseAxis : MXBaseAxisType;
	END_STRUCT;
	MXCDCType : STRUCT
		ArcTransSpd : LREAL := 100;
		SpdMode : UDINT;
		ContourViolation : UDINT;
		TransMode : UDINT;
		EntryMode : USINT;
		AcrToLine : BOOL;
	END_STRUCT;
	MXAutoTangType : STRUCT
		Offset : LREAL;
	END_STRUCT;
	MXHWTriggerType :	STRUCT
		Source : UINT;
		Index : UINT;
	END_STRUCT;
	MXTriggerConfigType : 	STRUCT
		Type : UINT;
		Edge : UINT;
		HWTrigger : MXHWTriggerType;
	END_STRUCT;
END_TYPE

(********************************************************************
 * COPYRIGHT (C) BERNECKER + RAINER, AUSTRIA, A-5142 EGGELSBERG
 ********************************************************************
 * Library: ARNC0MX
 * File: arnc0mx.fun
 * Created: 13.06.2012
 ********************************************************************
 * Functions and function blocks of library ARNC0MX
 ********************************************************************)
FUNCTION MXPointToJointEx1 : UDINT
	VAR_INPUT
		AddrTrfData : UDINT;
		Point : MXPointType;
		Joint : MXJointAxisType;
		TrfType : UDINT;
		Tool : MXToolType;
		BaseFrame : MXFrameType;
		RefJoint : ARRAY[0..5] OF LREAL;
	END_VAR
END_FUNCTION

FUNCTION MXPointToJointEx : UDINT
	VAR_INPUT
		AddrTrfData : UDINT;
		Point : MXPointType;
		Joint : MXJointAxisType;
		TrfType : UDINT;
		Tool : MXToolType;
		BaseFrame : MXFrameType;
		RefJoint : MXJointAxisType;
	END_VAR
END_FUNCTION

FUNCTION MXJointToPointEx1 : UDINT
	VAR_INPUT
		AddrTrfData : UDINT;
		Joint : MXJointAxisType;
		Point : MXPointType;
		AnglesType : UDINT;
		TrfType : UDINT;
		Tool : MXToolType;
		BaseFrame : MXFrameType;
		RefPath : ARRAY[0..5] OF LREAL;
	END_VAR
END_FUNCTION

FUNCTION MXJointToPointEx : UDINT
	VAR_INPUT
		AddrTrfData : UDINT;
		Joint : MXJointAxisType;
		Point : MXPointType;
		AnglesType : UDINT;
		TrfType : UDINT;
		Tool : MXToolType;
		BaseFrame : MXFrameType;
		RefPoint : MXPointType;
	END_VAR
END_FUNCTION

FUNCTION MXCncAxesToPoint : UDINT
	VAR_INPUT
		AddrTrfData : UDINT;
		Axis : ARRAY[0..14] OF LREAL;
		Point : MXPointType;
		TrfType : UDINT;
		AnglesType : UDINT;
		AxisMapCode : ARRAY[0..14] OF UINT;
		AxisMapIdx : ARRAY[0..14] OF UINT;
		ActiveAxesCount : UDINT;
	END_VAR
END_FUNCTION

FUNCTION MXFromOrient : UDINT
	VAR_INPUT
		Orient : MXOrientationType;
		Matrix : ARRAY[0..8] OF LREAL;
	END_VAR
END_FUNCTION

FUNCTION MXToOrient : UDINT
	VAR_INPUT
		Matrix : ARRAY[0..8] OF LREAL;
		Type : UDINT;
		Orient : MXOrientationType;
		RefAngle : ARRAY[0..2] OF LREAL;
	END_VAR
END_FUNCTION

FUNCTION MXConvertOrient : UDINT
	VAR_INPUT
		OrientIn : MXOrientationType;
		Type : UDINT;
		OrientOut : MXOrientationType;
		RefAngle : ARRAY[0..2] OF LREAL;
	END_VAR
END_FUNCTION

FUNCTION MXFrameRotX : UDINT
	VAR_INPUT
		Frame : MXFrameType;
		Angle : LREAL;
	END_VAR
END_FUNCTION

FUNCTION MXFrameRotY : UDINT
	VAR_INPUT
		Frame : MXFrameType;
		Angle : LREAL;
	END_VAR
END_FUNCTION

FUNCTION MXFrameRotZ : UDINT
	VAR_INPUT
		Frame : MXFrameType;
		Angle : LREAL;
	END_VAR
END_FUNCTION

FUNCTION MXFrameEuler : UDINT
	VAR_INPUT
		Frame : MXFrameType;
		Phi : LREAL;
		Theta : LREAL;
		Psi : LREAL;
	END_VAR
END_FUNCTION

FUNCTION MXFrameRPY : UDINT
	VAR_INPUT
		Frame : MXFrameType;
		Roll : LREAL;
		Pitch : LREAL;
		Yaw : LREAL;
	END_VAR
END_FUNCTION

FUNCTION MXFrameTrans : UDINT
	VAR_INPUT
		Frame : MXFrameType;
		DistanceX : LREAL;
		DistanceY : LREAL;
		DistanceZ : LREAL;
	END_VAR
END_FUNCTION

FUNCTION MXFrameTransX : UDINT
	VAR_INPUT
		Frame : MXFrameType;
		Distance : LREAL;
	END_VAR
END_FUNCTION

FUNCTION MXFrameTransY : UDINT
	VAR_INPUT
		Frame : MXFrameType;
		Distance : LREAL;
	END_VAR
END_FUNCTION

FUNCTION MXFrameTransZ : UDINT
	VAR_INPUT
		Frame : MXFrameType;
		Distance : LREAL;
	END_VAR
END_FUNCTION

FUNCTION MXFrameApply : UDINT
	VAR_INPUT
		Frame1 : MXFrameType;
		Frame2 : MXFrameType;
	END_VAR
END_FUNCTION

FUNCTION MXFromFrame : UDINT
	VAR_INPUT
		Frame : MXFrameType;
		PointIn : MXPointType;
		PointOut : MXPointType;
	END_VAR
END_FUNCTION

FUNCTION MXToFrame : UDINT
	VAR_INPUT
		Frame : MXFrameType;
		PointIn : MXPointType;
		PointOut : MXPointType;
	END_VAR
END_FUNCTION

(********************************************************************
 * COPYRIGHT -- Bernecker + Rainer
 ********************************************************************
 * Library: Motion Command Extension
 * File: arnc0mx.var
 * Author: B&R
 ********************************************************************
 * Constants of Motion Command Library
 ********************************************************************)

(* Velocity mode constants (<MXVelocityType>.Mode) *)
VAR CONSTANT
  MX_VEL_MODE_RAPID : UDINT := 0; (* rapid mode *)
  MX_VEL_MODE_FEED  : UDINT := 1; (* feedrate mode *)
  MX_VEL_MODE_TIME  : UDINT := 2; (* inverse time mode *)
END_VAR

(* MXVelocityType constants *)
VAR CONSTANT
  MX_VEL_RAPID  : MXVelocityType := (Mode:=0);           (* rapid movement         *)
  MX_VEL_F50000 : MXVelocityType := (v:=50000, Mode:=1); (* 50000 units per minute *)
  MX_VEL_F10000 : MXVelocityType := (v:=10000, Mode:=1); (* 10000 units per minute *)
  MX_VEL_F5000  : MXVelocityType := (v:=5000,  Mode:=1); (* 5000 units per minute  *)
  MX_VEL_F1000  : MXVelocityType := (v:=1000,  Mode:=1); (* 1000 units per minute  *)
  MX_VEL_F500   : MXVelocityType := (v:=500,   Mode:=1); (* 500 units per minute   *)
  MX_VEL_F100   : MXVelocityType := (v:=100,   Mode:=1); (* 100 units per minute   *)
END_VAR

(* Trigger configuration constants *)
VAR CONSTANT
  MX_TRIGGER_HW	            : UINT := 0;           (* Hardware trigger - MXHWTriggerType *)
  MX_TRIGGER_POSITIVE_EDGE  : UINT := 0;           (* Positive edge						 *)
  MX_TRIGGER_NEGATIVE_EDGE  : UINT := 1;           (* Negative edge						 *)
  MX_TRIGGER_HW_INPUT1		: UINT := 1;           (* Hardware trigger input 1			 *)
  MX_TRIGGER_HW_INPUT2		: UINT := 2;           (* Hardware trigger input 1			 *)
END_VAR

(* MXFrameMXFrameType constants *)
VAR CONSTANT
  MX_FRM_ZERO : MXFrameType := (0); (* zero (identity) frame *)
END_VAR

(* Transition type constants (<MXPathTransType>.Type) *)
VAR CONSTANT
  MX_TRANS_OFF      : UDINT := 0; (* Transition deactivated *)
  MX_TRANS_ACCURATE : UDINT := 1; (* Accuracy hold *)
  MX_TRANS_ARC      : UDINT := 2; (* Tangential transition arcs *)
  MX_TRANS_ROUND    : UDINT := 3; (* Rounding edges *)
END_VAR

(* Orientation type constants (<MXOrientationType>.Type) matches constants from TRF_LIB *)
VAR CONSTANT
  MX_CARDAN_XYZ_ANGLES    : UDINT := 1;      (* Cardan XYZ angles *)
  MX_EULER_XYZ_ANGLES     : UDINT := 1;      (* Cardan XYZ angles *)
  MX_CARDAN_XZY_ANGLES    : UDINT := 2;      (* Cardan XZY angles *)
  MX_EULER_XZY_ANGLES     : UDINT := 2;      (* Cardan XZY angles *)
  MX_CARDAN_YXZ_ANGLES    : UDINT := 4;      (* Cardan YXZ angles *)
  MX_EULER_YXZ_ANGLES     : UDINT := 4;      (* Cardan YXZ angles *)
  MX_CARDAN_YZX_ANGLES    : UDINT := 8;      (* Cardan YZX angles *)
  MX_EULER_YZX_ANGLES     : UDINT := 8;      (* Cardan YZX angles *)
  MX_CARDAN_ZXY_ANGLES    : UDINT := 16;     (* Cardan ZXY angles *)
  MX_EULER_ZXY_ANGLES     : UDINT := 16;     (* Cardan ZXY angles *)
  MX_CARDAN_ZYX_ANGLES    : UDINT := 32;     (* Cardan ZYX angles *)
  MX_EULER_ZYX_ANGLES     : UDINT := 32;     (* Cardan ZYX angles *)
  MX_EULER_XYX_ANGLES     : UDINT := 64;     (* Euler XYX angles  *)
  MX_EULER_XZX_ANGLES     : UDINT := 128;    (* Euler XZX angles  *)
  MX_EULER_YXY_ANGLES     : UDINT := 256;    (* Euler YXY angles  *)
  MX_EULER_YZY_ANGLES     : UDINT := 512;    (* Euler YZY angles  *)
  MX_EULER_ZXZ_ANGLES     : UDINT := 1024;   (* Euler ZXZ angles  *)
  MX_EULER_ZYZ_ANGLES     : UDINT := 2048;   (* Euler ZYZ angles  *)
  MX_POSITIVE_ANGLES      : UDINT := 4096;   (* mathematically positive angles *)
  MX_NEGATIVE_ANGLES      : UDINT := 8192;   (* mathematically negative angles *)
  MX_DIRECT_ANGLES        : UDINT := 16384;  (* direct "R" rotation matrix     *)
  MX_INDIRECT_ANGLES      : UDINT := 32768;  (* indirect "R^T" rotation matrix *)
  MX_EULER_ANGLES         : UDINT := 1024;   (* Euler ZXZ is commonly in view  *)
  MX_CARDAN_ANGLES        : UDINT := 1;      (* Cardan XYZ is commonly in view *)
  MX_NAUTICAL_ANGLES      : UDINT := 1;      (* Cardan XYZ is commonly in view *)
  MX_TAIT_BRYAN_ANGLES    : UDINT := 1;      (* Cardan XYZ is commonly in view *)
  MX_QUATERNION           : UDINT := 8000;   (* quaternion *)
END_VAR

(* Kinematics configuration mode constants (<MXConfigType>.Mode) matches constants from TRF_LIB *)
VAR CONSTANT
  MX_MODE_FRONT           : UDINT := 1;          (* front *)
  MX_MODE_BACK            : UDINT := 2;          (* back *)
  MX_MODE_CONVEX          : UDINT := 4;          (* convex *)
  MX_MODE_CONCAVE         : UDINT := 8;          (* concave *)
  MX_MODE_POSITIVE        : UDINT := 16;         (* positive *)
  MX_MODE_NEGATIVE        : UDINT := 32;         (* negative *)
  MX_MODE_LEFT            : UDINT := 64;         (* left *)
  MX_MODE_RIGHT           : UDINT := 128;        (* right *)
  MX_MODE_DIRECT          : UDINT := 256;        (* direct *)
  MX_MODE_INDIRECT        : UDINT := 512;        (* indirect *)
  MX_MODE_CONVEX2         : UDINT := 1024;       (* convex2 *)
  MX_MODE_CONCAVE2        : UDINT := 2048;       (* concave2 *)
  MX_MODE_CONVEX3         : UDINT := 4096;       (* convex3 *)
  MX_MODE_CONCAVE3        : UDINT := 8192;       (* concave3 *)
  MX_MODE_HETEROGENEOUS   : UDINT := 16384;      (* heterogeneous *)
  MX_MODE_HOMOGENEOUS     : UDINT := 32768;      (* homogeneous *)
  MX_MODE_LEFT2           : UDINT := 65536;      (* left2 *)
  MX_MODE_RIGHT2          : UDINT := 131072;     (* right2 *)
  MX_MODE_NEG_DIR         : UDINT := 268435456;  (* negative direction forced *)
  MX_MODE_POS_DIR         : UDINT := 536870912;  (* positive direction forced *)
  MX_MODE_IN_SW_ENDS      : UDINT := 1073741824; (* in SW ends *)
END_VAR

(* Cutter diameter compensation constants *)
VAR CONSTANT
  MX_CDC_LEFT                    : UDINT := 0;      (* CDC left *)
  MX_CDC_RIGHT                   : UDINT := 1;      (* CDC right *)
  MX_CDC_SPD_ON_CONTOUR          : UDINT := 0;      (* Path speed moves to the contour *)
  MX_CDC_SPD_ON_TCP              : UDINT := 1;      (* Path speed moves to the center of the tool *)
  MX_CDC_NO_COUNTER_VIOLATION    : UDINT := 0;      (* Do NOT allow contour violations due to very short path *)
  MX_CDC_VIOLATION_SHORT_PATH    : UDINT := 1;      (* Allow contour violations due to very short path sections *)
  MX_CDC_VIOLATION_INNER_EDGE    : UDINT := 2;      (* Allow contour violations due to an inner edge without intersection *)
  MX_CDC_LINEAR_TRANSITION       : UDINT := 0;      (* CDC with linear transitions *)
  MX_CDC_ARC_TRANSITION          : UDINT := 1;      (* CDC with arc transitions *)
  MX_CDC_ENTRY_BLOCK             : UDINT := 0;      (* Activate/deactivate CDC indirectly with transi-tion block *)
  MX_CDC_ENTRY_DIRECT            : UDINT := 1;      (* Activate/deactivate CDC directly *)
  MX_CDC_ENTRY_INDIRECT          : UDINT := 2;      (* Activate/deactivate CDC indirectly *)
  MX_CDC_NO_ARC_TO_LINE          : UDINT := 0;      (* Deactivate replacement of arc with straight line *)
  MX_CDC_ARC_TO_LINE             : UDINT := 1;      (* Activate replacement of arc with straight line *)
END_VAR

(* Transformation function types *)
VAR CONSTANT
  MX_TRF_TYPE_INVERSE            : UDINT := 0;      (* TRF_inverse  function *)
  MX_TRF_TYPE_INVERSE2           : UDINT := 1;      (* TRF_inverse2 function *)
  MX_TRF_TYPE_INVERSE3           : UDINT := 2;      (* TRF_inverse3 function *)
  MX_TRF_TYPE_DIRECT             : UDINT := 0;      (* TRF_direct   function *)
  MX_TRF_TYPE_DIRECT2            : UDINT := 1;      (* TRF_direct2  function *)
  MX_TRF_TYPE_DIRECT3            : UDINT := 2;      (* TRF_direct3  function *)
END_VAR

(* Statuses, warnings, errors *)
VAR CONSTANT
  MX_OK                          : UDINT := 0;     (* Status OK *)
  MX_WARNING_AXES                : UDINT := 2001;  (* Transformation returns valid values with warnings on axes *)
  MX_WARNING_REF_POINT_ANGLES    : UDINT := 2002;  (* Values in reference point or reference joint axes may be ignored due to conversion to another angles type *)
  MX_ERROR_WRONG_ANGLE_TYPE      : UDINT := 6001;  (* Angles type is not supported *)
  MX_ERROR_TRF_DATA_NOT_DEFINED  : UDINT := 6002;  (* Address of the transformation data variable is zero *)
  MX_ERROR_WRONG_ROBOT           : UDINT := 6003;  (* Robot is not supported *)
  MX_ERROR_WRONG_TRF_TYPE        : UDINT := 6004;  (* Transformation type not supported *)
  MX_ERROR_TRF_LIB_NOT_SUPPORTED : UDINT := 6005;  (* Transformation library of not supported version *)
  MX_ERROR_TRF_CMD_CODE			 : UDINT := 8001;  (* Unknown command code *)
  MX_ERROR_TRF_MEASURE           : UDINT := 8002;  (* Unknown measure *)
  MX_ERROR_TRF_ANGLES_TYPE       : UDINT := 8003;  (* Unknown angles type *)
  MX_ERROR_TRF_GEN29_CMD_CODE    : UDINT := 9001;  (* Unknown command code *)
  MX_ERROR_UNKNOWN_ROBOT         : UDINT := 9002;  (* Unknown robot *)
  MX_ERROR_INVALID_TRF_TYPE      : UDINT := 9003;  (* Invalid type of transformation *)
  MX_ERROR_TRF_ERROR_AXES        : UDINT := 10003; (* Transformation function returns error of axis *)
  MX_ERROR_TRF_NOT_LICENSED      : UDINT := 10008; (* Transformation function not licenced *)
  MX_ERROR_TRF_NOT_SUPPORTED     : UDINT := 10009; (* Transformation function not supported *)
  MX_ERROR_FCT_NOT_DEFINED       : UDINT := 10010; (* Transformation function address is zero *)
  MX_ERROR_TRF_INVALID_INPUTS    : UDINT := 10015; (* Invalid inputs for transformation error *)
END_VAR

(* Error offsets *)
VAR CONSTANT
  MX_OFFSET_WARNING              : UDINT := 2000;  (* ARNC0MX warnings *)
  MX_OFFSET_WARNING_TRF_FUN      : UDINT := 4000;  (* TRF_LIB warnings *)
  MX_OFFSET_ERROR                : UDINT := 6000;  (* ARNC0MX errros *)
  MX_OFFSET_ERROR_TRF_FUN        : UDINT := 12000; (* TRF_LIB errors *)
END_VAR

(********************************************************************
 * COPYRIGHT -- Bernecker + Rainer
 ********************************************************************
 * Library: Motion Command Library
 * File: arnc0mxsv.var
 * Author: B&R
 ********************************************************************
 * System Variables of Motion Command Library
 ********************************************************************)
VAR {SHARED_IP_GLOBAL}
   _Frm  : MXFrameType;
   _Tool : MXToolType;
   _Vel  : MXVelocityType;
   _Base : MXFrameType;
   _Ref  : MXJointAxisType;
   _Pth  : MXPathDescType;
   _Dyn  : MXDynamicDescType;
END_VAR

VAR CONSTANT
   FRM_0   : MXFrameType := (0);
   POINT_0 : MXPointType := (0);
   BASE_0  : MXFrameType := (0);
   TOOL_0  : MXToolType  := (0);
   VEL_0   : MXVelocityType := (Mode:=1);
   REF_0   : MXJointAxisType := (0);
   VEC6_0  : ARRAY[0..5] OF LREAL := 6(0.0);
   PTH_0   : MXPathDescType := (0);
   DYN_0   : MXDynamicDescType := (Accel:=100, Decel:=100);
   AXIS_TARGET_0 : MXAxisTargetType := (0);
END_VAR

VAR {SHARED_IP_GLOBAL}
  __tmp_point : MXPointType;
  __tmp_frame : MXFrameType;
  __tmp_tool : MXToolType;
  __tmp_vel : MXVelocityType;
  __tmp_joint_axis : MXJointAxisType;
  __tmp_axis_target : MXAxisTargetType;
  __tmp_pth : MXPathDescType;
  __tmp_dynamic : MXDynamicDescType;
  __tmp_cdc : MXCDCType;
  __tmp_auto_tang : MXAutoTangType;
  __tmp_trigger : MXTriggerConfigType;
  __mx_status : UDINT;
  __tmp_vec6 : ARRAY[0..5] OF LREAL;
  __tmp_set_pos : ARRAY[0..14] OF LREAL;
  __tmp_axis_code : ARRAY[0..14] OF UINT;
  __tmp_axis_idx : ARRAY[0..14] OF UINT;
END_VAR
```

### gmcipsys.cnc
```
LANGS (defaultLangId=1, defaultDataLangId=3)
  CMDQUEUE (BufferSize=15)
  MEM (ReserveMB=5, LimitPercent=80%)
  EXEC (InstrBurstBG=200, CycleBurstBG=0, Stack=16384, MinorStack=2048, EStack=1024)
  LOAD (ReadLineBurstMax=100, ReadLineBurstMin=20, ParseLineBurstMax=10, ParseLineBurstMin=2, RuntimeIOBlocking=No)
  DISABLE_MSG = 15238 
    15336 
    15337 
    15666 
    15784 
    15864 
    15740
  LANG (langId=1, langName=B&R GCode, langModule=ailgcode)
    LANGCONFIG gmciplbr
    LANGCONFIG gmcipcbr
    LANGCONFIG gmcipubr
    FILEEXT .cnc
    FILEEXT .prg
    MAINSEARCHPATH $ (FileDevice=CNC_PrgDir)
    MAINSEARCHPATH $ (DataObject=Yes)
    INCLUDEPATH $ (FileDevice=CNC_PrgDir)
    INCLUDEPATH $ (DataObject=Yes)
  LANG (langId=2, langName=Alternative Language 1 GCode, langModule=ailgcode)
    LANGCONFIG gmciplsm
    LANGCONFIG gmcipcbr
    LANGCONFIG gmcipcsm
    LANGCONFIG gmcipusm
    FILEPREFIX = _N_
    FILEEXT = .MPF
    FILEEXT = _MPF
    FILEEXT = .SPF
    FILEEXT = _SPF
    MAINSEARCHPATH = \$ (FileDevice=CNC_PrgDir)
    MAINSEARCHPATH = \_N_MPF_DIR\$ (FileDevice=CNC_PrgDir)
    MAINSEARCHPATH = \_N_SPF_DIR\$ (FileDevice=CNC_PrgDir)
    MAINSEARCHPATH = $ (DataObject=1)
    INCLUDEPATH = \$ (FileDevice=CNC_PrgDir)
    INCLUDEPATH = \_N_SPF_DIR\$ (FileDevice=CNC_PrgDir)
    INCLUDEPATH = \_N_MPF_DIR\$ (FileDevice=CNC_PrgDir)
    INCLUDEPATH = $ (DataObject=1)
  LANG (langId=3, langName=IEC-ST, langModule=ailgcode)
    LANGCONFIG gmcipiec
    LANGCONFIG gmcipmx (RequireFnIgnore=MXConvertOrient)
    LANGCONFIG gmcipui (IfNotExist=Warn)
    FILEEXT .typ (DeclScope=IP_GLOBAL)
    FILEEXT .var (DeclScope=IP_GLOBAL)
    FILEEXT .fun (DeclScope=IP_GLOBAL)
    FILEEXT .iec (DeclScope=IP_LOCAL)
    FILEEXT .st (DeclScope=IP_LOCAL)
    FILEEXT _iec (DeclScope=IP_LOCAL)
    MAINSEARCHPATH = \$ (FileDevice=IEC_PrgDir)
    MAINSEARCHPATH = \$ (FileDevice=CNC_PrgDir)
    MAINSEARCHPATH \TYP\$ (FileDevice=CNC_PrgDir, DataObject=No)
    INCLUDEPATH = \$ (FileDevice=IEC_PrgDir)
    INCLUDEPATH = \$ (FileDevice=CNC_PrgDir)
    INCLUDEPATH \TYP\$ (FileDevice=CNC_PrgDir, DataObject=No)
  XML_INCLUDE gmcipus (IfNotExist=Warn)
```

- Data object Logical/GmcIpUserConfig/gmcipfun (Cnc, version 3.13.0) (no source held here)

- Data object Logical/GmcIpUserConfig/gmcipfub (Cnc, version 3.13.0) (no source held here)

- Data object Logical/GmcIpUserConfig/gmcipubr (Cnc, version 3.13.0) (no source held here)

- Data object Logical/GmcIpUserConfig/gmcipusm (Cnc, version 3.13.0) (no source held here)

- Data object Logical/GmcIpUserConfig/gmcipui (Cnc, version 3.13.0) (no source held here)

- Data object Logical/GmcIpUserConfig/gmcipus (Cnc, version 3.13.0) (no source held here)

- Data object Logical/GmcIpUserConfig/gmcipuc (Cnc, version 3.13.0) (no source held here)

### Data object Logical/CncInit (Cns)

- CncInit.cns (not shown)

### Data object Logical/CncProg (Cnc)

#### CncProg.cnc
```
%001 (CncProgram)
```

### Program Logical/SDCAxisCtr (ANSIC)

#### Main.c
```c
#include <bur/plctypes.h>

#ifdef _DEFAULT_INCLUDES
	#include <AsDefault.h>
#endif

void increase_counters(void);

void _INIT ProgramInit(void)
{
	//Устанваливаем типы SDC модулей
	AxisX_HW.EncIf1_Typ = ncSDC_ENC16;
	AxisX_HW.DiDoIf_Typ = ncSDC_DIDO;
	AxisX_HW.DrvIf_Typ = ncSDC_DRVSERVO16;

	//Устанавливаем имена переменных
	strcpy(AxisX_HW.EncIf1_Name, "AxisX_EncIf");
	strcpy(AxisX_HW.DrvIf_Name, "AxisX_DrvIf");
	strcpy(AxisX_HW.DiDoIf_Name, "AxisX_DiDoIf");

	//Устанавливаем входы готовности и нормальной работы
	AxisX_EncIf.iEncOK = 1;
	AxisX_DrvIf.iDrvOK = 1;
	AxisX_DrvIf.iStatusEnable = 1;
	AxisX_DiDoIf.iDriveReady = 1;

	fb_controller.dt = 0.002;
	fb_controller.k_i = 0.16;
	fb_controller.k_p = 0.0064;
	fb_controller.max_abs_value = 24.0;

	pwm_period = 200;
}

void _CYCLIC ProgramCyclic(void)
{
	FB_Axis(&axis_X);
	coil_pwm_value = coil_powered ? 32767 : 0;

	increase_counters();

	//Формирование показаний датчика

	AxisX_EncIf.iActTime = (INT)	AsIOTimeCyclicStart();
	AxisX_EncIf.iActPos = axis_X.counter;
	AxisX_DiDoIf.iPosHwEnd = axis_X.endswitch_b_reached;
	AxisX_DiDoIf.iNegHwEnd = axis_X.endswitch_a_reached;
	fb_controller.in = AxisX_DrvIf.oSetPos;

	if((fb_controller.in<min_task)&&(fb_controller.in>(-min_task))) fb_controller.in = 0;
	fb_controller.in = fb_controller.in * 6500/32767 - axis_X.speed;

	FB_Controller(&fb_controller);

	axis_X.pwm_value = fb_controller.out / 24.0 * 32767;
}

void increase_counters(void)
{
	AxisX_EncIf.iLifeCnt++;
	AxisX_DiDoIf.iLifeCntDriveEnable++;
	AxisX_DiDoIf.iLifeCntDriveReady++;
	AxisX_DiDoIf.iLifeCntNegHwEnd++;
	AxisX_DiDoIf.iLifeCntPosHwEnd++;
	AxisX_DiDoIf.iLifeCntReference++;
	AxisX_DrvIf.iLifeCnt++;
}

void _EXIT ProgramExit(void)
{
	// Insert code here

}
```

### Program Logical/SDCAxisCtr1 (ANSIC)
